(* CoDeSys 2.3 project: cy-wg-018-00.pro *)
(* Title: cy-wg-06 - ClevergyAS *)
(* Author: Andrea Ravasio *)
(* Libraries: Standard.lib 2.12.10 14:48:34, Util.lib 26.9.14 10:12:46, Visual.lib 2.12.10 14:48:34, WagoLibIdent.lib 25.2.13 11:12:16, WagoLibStatus.lib 2.12.10 14:48:32, SysLibFile.lib 2.12.10 14:48:34, SysLibRtc.lib 2.12.10 14:48:32, SysLibSockets.lib 10.2.11 09:20:54, SysLibEvent.lib 2.12.10 14:48:34, SysLibPlcCtrl.lib 2.12.10 14:48:32, SysLibCallback.lib 2.12.10 14:48:32, mod_com.lib 2.12.10 14:48:32, SerComm.lib 31.5.11 08:54:36, Serial_Interface_01.lib 22.4.13 12:50:14, Modb_l05.lib 22.4.13 12:50:12, Ethernet.lib 2.12.10 14:48:32, MBus_03.lib 22.7.15 16:25:47, WagoLibModbus_IP_01.lib 24.7.13 15:05:58, WagoLibMBX_01.lib 20.3.12 16:32:40, LON_01.lib 22.7.15 16:25:47 *)

(* PLC configuration (modules and I/O channels)
0750-9999/0545-0008 8 DO/DI Generic [Type_34_8_Channels] node 0, in %IB68 out %QB44 {INTTypePAAssignment = PLC; INTTypeModule = plugged}
  VPN_ST2 AT %IX34.0 [BOOLOnX_I] I 1: Digital Input
  LAMP_AL AT %QX22.0 [BOOLOnX_Q] I 2: Digital Input
  KEY_QE_ST AT %IX34.1 [BOOLOnX_I] I 3: Digital Input
  CIR01_EN AT %QX22.1 [BOOLOnX_Q] I 4: Digital Input
  CIR01_AL AT %IX34.2 [BOOLOnX_I] I 5: Digital Input
  CIR04_EN AT %QX22.2 [BOOLOnX_Q] I 6: Digital Input
  CIR01_ST AT %IX34.3 [BOOLOnX_I] I 7: Digital Input
  CAL01_EN AT %QX22.3 [BOOLOnX_Q] I 8: Digital Input
  CIR01_AUTO AT %IX34.4 [BOOLOnX_I] O 0: Digital Output
  CAL01_RST AT %QX22.4 [BOOLOnX_Q] O 1: Digital Output
  CIR04_AL AT %IX34.5 [BOOLOnX_I] O 2: Digital Output
  AT %QX22.5 [BOOLOnX_Q] O 3: Digital Output
  CIR04_ST AT %IX34.6 [BOOLOnX_I] O 4: Digital Output
  AT %QX22.6 [BOOLOnX_Q] O 5: Digital Output
  CIR04_AUTO AT %IX34.7 [BOOLOnX_I] O 6: Digital Output
  AT %QX22.7 [BOOLOnX_Q] O 7: Digital Output
0750-9999/0400-0008 8 DI Generic [Type_1_8_Channels] node 1, in %IB68 out %QB44 {INTTypePAAssignment = PLC; INTTypeModule = plugged}
  CIRD01_A_AUTO AT %IX34.8 [BOOLOnX_I] Ch_1 Digital input
  CIRD01_B_AL AT %IX34.9 [BOOLOnX_I] Ch_2 Digital input
  CIRD01_A_AL AT %IX34.10 [BOOLOnX_I] Ch_3 Digital input
  CTL01_ST AT %IX34.11 [BOOLOnX_I] Ch_4 Digital input
  CIR02_AL AT %IX34.12 [BOOLOnX_I] Ch_5 Digital input
  CIRD01_B_AUTO AT %IX34.13 [BOOLOnX_I] Ch_6 Digital input
  CAL01_AL AT %IX34.14 [BOOLOnX_I] Ch_7 Digital input
  CAL01_ST AT %IX34.15 [BOOLOnX_I] Ch_8 Digital input
0750-9999/0400-0008 8 DI Generic [Type_1_8_Channels] node 2, in %IB69 out %QB45 {INTTypePAAssignment = PLC; INTTypeModule = plugged}
  CIR02_AUTO AT %IX35.0 [BOOLOnX_I] I 1: Digital Input
  AT %IX35.1 [BOOLOnX_I] I 2: Digital Input
  AT %IX35.2 [BOOLOnX_I] I 3: Digital Input
  CIR03_AL AT %IX35.3 [BOOLOnX_I] I 4: Digital Input
  CIR03_AUTO AT %IX35.4 [BOOLOnX_I] I 5: Digital Input
  AT %IX35.5 [BOOLOnX_I] I 6: Digital Input
  AT %IX35.6 [BOOLOnX_I] I 7: Digital Input
  AT %IX35.7 [BOOLOnX_I] I 8: Digital Input
0750-0464#04 2/4 AI RTD / ADJ./ HA [Type_44_4_Channels] node 3, in %IB64 out %QB40 {INTTypePAAssignment = PLC; INTTypeModule = plugged}
  S01 AT %IW0 [INTOnW_I] Channel 1
  S02 AT %IW1 [INTOnW_I] Channel 2
  S03 AT %IW2 [INTOnW_I] Channel 3
  AT %IW3 [INTOnW_I] Channel 4
0750-0464#04 2/4 AI RTD / ADJ./ HA [Type_44_4_Channels] node 4, in %IB64 out %QB40 {INTTypePAAssignment = PLC; INTTypeModule = plugged}
  S05 AT %IW4 [INTOnW_I] Channel 1
  S07 AT %IW5 [INTOnW_I] Channel 2
  S06 AT %IW6 [INTOnW_I] Channel 3
  S08 AT %IW7 [INTOnW_I] Channel 4
0750-0464#04 2/4 AI RTD / ADJ./ HA [Type_44_4_Channels] node 5, in %IB72 out %QB40 {INTTypePAAssignment = PLC; INTTypeModule = plugged}
  S09 AT %IW8 [INTOnW_I] Channel 1
  S11 AT %IW9 [INTOnW_I] Channel 2
  S10 AT %IW10 [INTOnW_I] Channel 3
  S12 AT %IW11 [INTOnW_I] Channel 4
0753-0648 LON-FTT [Type_55_1_Channels] node 6, in %IB80 out %QB40 {INTTypePAAssignment = PLC; INTTypeModule = plugged; DataStream = 1F8B0800000000000400ED5D7B6FE2C8B2FFFF4AF73BF820DDD5AC14261808796C921503668296470E8FCC8E6646C88106BC636C8E1FC9E47CFA5BD56D1B1BB71F0498248CA5D52CB1DBD555DDD5BF7A74B97DF9E78F852A3C10C35474ED2A27BE2FE404A28DF589A2CDAE72B635CD8B95DC9FD7FFFB3F972D5D6B6A1631A6; DataStream = F29808F090665EFC3095ABDCDCB29617C7C78F8F8FEF1F4BEF7563765C2C14C4E3BFDBADFE784E16725ED14C4BD6C624E73D35497E2A27DC1AFACC90174D687C5EB828142E4EE1DF938B827851A85C14CAF02327FCAD4C3BF2825CE5DAB6A68C95A5A2D78949B4FFCA9A9E13FA449DD6F5B1BD209A255B205E4D5FE0EFAB5C; DataStream = 7532119E74DB10C6EC8A302706B0D721B6A16B0DC5583CCA06B9F3C6E49C76D4971FC8AD6CCDAF72B58BAF4313EE7E95B58941E4F7AAAC68CA57E8F9BBA52F73425B9FD82AE9D88B7B62C0D339183C41C0E16BCBC6F7EEFD3F646C99F4DAFA55E7225C1E90C552952DD29C0077CA542186770FEEE2C83427D78582C0FBEFF2; DataStream = D8B9EF7BA23FD697E41A6EB11FBE3B7F9127BC8EFFF35D6D6A13F2E35ABC3C663F3CBE8E6318F398C619B9EE376E079A3E214CB2D583F4A6F708B769B049D750668A26ABDCA6819BDE234DB3A58FBF93C9B565D8046470FFF43568C3D4C9966E3C796D56577CCDBA4BD41B59BD9ECAAA499B7957BC566D8213CDA61B8732F0; DataStream = B7D74A52096A5A4DB741DD60DD5C688A7A95C3CE73C2B16F4088F5A81BDFEF644391EF5562FA2765ED9EEF5692C63C4F6BE235C7D39EF3E2BAFAF854086F067528518F38BAD4B91B8CF4FB7F4606F98F4DCC286D5A6994F6A0F4DCA6E12601A5F137E56A532A8DDA40ABD26B5658BBC408EDA22DD3691823AA687DA24D06CA; DataStream = 824EADFFCF603BF947A09DEFCFF5763D3226CA03F135F55F5913FED6507443B19E56C27B57022DFBC47850C664F0049A571D7FD7F447954C666402DAE8BB1378A4AE18800C3090D74D6D69C3A4AE2E0459060B3755C63837D71D5D0326FC57024D6BBA365566B6416D08AC9225312C8598EB83DA34BDAED69465FD7AE0B10F; DataStream = 4F16E92BFF25D7A5CB63EFB76FD51F472FFB578B08A5384428ED1211C0B3B06C330520E87DA765221E782D5F3D1C143338480F075DDB7A5B785039183C388DC383D39DE1C1545109BA0869DC8306B4ED61D364F7C06BBA433CF0143D19105C9229F0E024C383C3750FC4E2E1E041390E0FCA3BC583F40E02AE7334FD695C84; DataStream = 55DB570F0A950C140ED849289E1E0C2A9C87D2506C8458D450D8292A2CF53490404DFFAD9E266858357DF580709A01C2E17A099B060DA13BAB8C6322CB97C7BCECF5F352DAF109EABC1891A1CE6F98A2A68BF24E312C5B5685A9AD8DD96A11EE5518D4F5CCF34669E498B59AE591D3E1FFEBCB2343F3B479E430ED1486C0D3; DataStream = 861D5A824D1248515A465B66A640786DBEA1275E96516623F4721965689D32A31CA29C01C36101C3CBFB881BE2C2E16496CFE23249673BCB2459A05AB87C17CB34B8808AD827295D063FE90C180E0B18DE9EC77038D9A4B3B3386438DB1532C8AA6C2CD2804295354C03090ECD0C0D0E0B0DDE9C9B503CCFD0609F6890DA47; DataStream = C800E12001E1EDB907878408711985B39D651430E627A9F28CEA539FB54D83080ED90C110E0B11DE9E8B7030782016E25C047A773788307F90C7A3853E49850A37B59A3882594E9F4FF091CFD0E1B0D0E1EDF90B62060F3F071E326CF8C5B1E1CD790E87040D27B1D070B2B35D08B8324AB5034171019BA5DF86706867B870; DataStream = 58B8F0F67C86430A295E2F3064A8F02BA3C29BF3163250D83728F4EDE53203865F1D183277214B313883B40287629681CCE0E18DC2C321A5195E353C64D8F08B63C39B8B290E091A5E634C51CC3290192EBC459FE190428AD70B0C192AFCCAA8F0E6BC850C14F60D0A5906320386CC5DC8520CDE20ADC0A1946520337878A3; DataStream = F070486986570D0F1936FCE2D8F0E6628A438286D7185394B20C64860B6FD16738A490E2F50243860ABF322ABC396F2103857D83429681CC80217317B2148337480E38D46F3E6509C80C1DDE283A6459863DFA0D080DD5B195790DBF3A2E64E144060B4158006FE15657B42CF9F84BE3C2DBF3173260D83330649B12192E64; DataStream = FEC2CBC1C2791C2A9CEF0C14CC47C51ACFD38042AD51476F41D27094521E00E910CF60E1B060217317325C08E0C2C70C17325CC8DC856C4FC21DA4A0CF90153E66E0F0069D866C4F628F390684866C43E2570785CC63C83021E42E641B12BF3C2EBC3D67210386FD0343E62FFCEAB870F0FE42E88EB9BA95C4F3E5714BD7DA; DataStream = B2F1BD7BFF0FB046AFAE5D33AF2FFFF5A556AF0EAA5F2EFFFCB1508507629840ED2A27BE2FE404A28D61C0B4D955CEB6A679B192FBF3FAB2265BB2AACFAE2F1B8A4A84A609FFB3884126F0484EA8C3CD3B8F44196960339CC2AB1CFE0B7FEBC642B6BC46156CD396FFD10DDF7339E156B6E657B9DAC557442D435E5032A6F0; DataStream = EEC759E5F7AF20C2271812F32B5234BFF607D54EBDDAABBF1F7CBE852729CC5DE522703027F4C814F8D5C624B615AA741FBF700BFC148FC5D271B1201605F1ECA258B8108BB9EB75B4A6AC70AF0A1F64D319813EACD4B1F5A5F22D27D0250CE2E7040A9E57B9D3524E4058BACAD18135C87F6C625A70EDC1620F238E8184D2; DataStream = A83FE80D6B0326290C0D8CA632664F52AC9BC2E323783C27A09621FB3961A829D0D96FAAF547537B90556522989601130BDD98BA6D8CC96F33EB0FBE503EF625CD5E082E79E46E64E1DCFD5016F6828A0220C37EE74557985EB41C5267D8E649E189DE57669AA3588E28AE2453DF10091A3C65E604E48EB0C5E00CE9098262; DataStream = 824C43CDA4BD804ECD602ECCA666911931685F4DB33FC6CF18D23F56729E9C944E5CF1684F3CE1869D7EF36347AA8F5ADDCEC79CD09D4E4D62514261811546043B23559FB8C580B84EAB7D4BE440BA60C102D06DEEC445C856E24F262537F2C8454BB950545531C958D726662A3961A6BF94566BC95B4075D00AB0F2A80982; DataStream = 3C99808E9B7C319ADDCE8AFD131EFB13D4728F0663F8C465D8C521AF9394EBBFB8E2B9E8F25C6524040B1F03E0B58CA7B8B51FCB34B263B9DC965C6E793DA4D5A5FE5C478A6994A954F2E140A914928F1A81189DEADF747B49023222214DF2E0E12C7FAF5882ED302F00E2310769BF2B2738C0CA86C85079163288952851D7; DataStream = 1D07EA463DC73E39A6C5BED78895D7F409895B53A9F4D3D4A29792C9E9670F5A2AFA94547C4B3AFA41B1BCC95913C8013F7D212B1A8FFD0FCD412341DF26CEC3D16C7B13C59A6E6C958453818A00FFF86CA223D0A95FA0E2A92B520794E1990269F4D16871A89E6934D2DA4488724888B22744D92F84CFAC02DE0A636C922C; DataStream = CA29DF92529B10230B1543D0A7023655483A23FA6C890686AC99320D79A8B36024CB75C65D283F46CEE3D1A2D106307A30599B82F906A0503C3909C2DD262070CE453A874CB464AC855F05B700EED36FFEA5C458F868E8F6726BC89E2DA3217B16E8616B004B42E1A04A3D0B7BEF755D25B2B60FD8AAAC5408FA7C26FF267D; DataStream = 340508B3A167CD7F79D3C1F8186AB6096DA70A5127CF14C5A624E244498AA4335392999200006F6D49668CCA762AC9372DCF3138CF73B91D80B7AD39EE098C5984AE7311276A70C40237E20592233D167D36C7FCE7C8E6E6B837958A9B175A02B10DA4DAC271287FF3AF503723590E64244D4BB6EC580F222E21E93EEDC4AF; DataStream = A7BBCF49B21E02294951E4E624FB919244A52457DCC7662459B3E8846465FF49888E87DCC85144DE2B7D6A921982913E1D39E4A253118E41DAB7807DA292B1452DBC1A1FA5A7C84E9A0EB11123B6B30C2C662663B27CCFCD46CA13C3E36C67597D07022212A96343595A3AD720A70A1C263E12BBE6BC6A18F2D317B1F20DD5; DataStream = BDC16668AA0B325E1608DB2A5D79BCB8D562D2477C78ED3DC513B0DAEB553F27C847A187117010A1E28AC7F800D6C48A309ECB063838C4489124A6ABA3060FA4B43D08A63E942B9E85845B1F12CE5CB22553BBA9F6560217B9B6D693F88B78F26D6DCD44A1234B7655FBB566733514CF375AB49F7FDBF224A53326964FCB67; DataStream = A54AF93429367386E1DFC36ADD370C5C64E4C4686BD2973D23FD646DE4413F1319074969CB20201637099D53AFD99D3A2289A0997A3BC4B77D73BE5BF861E8C34267A1598F401F2EF8780F3D177C58203D5226AE6C61ECA9084CFBF61BE3448ABFAD63EF49F8258435E9B2E93F29B8A9AC8D844AB49935DF3E0470E477C945; DataStream = 0F80D411C4F279E12C2FBAE915F799579729C58284DDA44A771FC7256F3A444AC5753037DD7FD82442DF026645DF169FB8AA41392BF94324223C80731CEFFB45847C180811CE6625BAD0CA8332B16555C0054BD7E90E72C68C5DA458884E1D857985070ABBC91944272613F81537E457DC0FBFC5B4FC1637E4B7B81F7E4B69; DataStream = F92D6DC86F693FFC96D3F25BDE90DFF27EF83D49CBEFC986FC9EEC87DF4A5A7E2B1BF25BD90FBFA769F93DDD90DFD31DF29B8EC3B3E4643DD7B58167CF5E187CCF9FCFFAF90BE3B01863E8927817F764F45283B21863F51299DF93054C8DD0628C094C647E4FE630355C8B31F63091F93DD9C6D4D82DC618C744E6F7642853; DataStream = 03B918632913994F6D357756F5E746045E16060BE2718363C1DDCB4C880770D375E43CCCB8F736809E886C1C090B5DB3E647C2447E3A12E6BA8D5714CDB6C891C00A8253664DD367CE4A05ACF2E76C0E7D26323FE2F1E7D0C2623ED1C7E2D28145BFC49BA403378A5F5D31DA38A09BC4AFDCA07CC1A844EB1E6DB027614AAB; DataStream = 4499CC2D868E12851B894FE4D88A07B8BD27318A5E507D038ABD891C659E1C734A245A10BCBF27494ECE3DEDA28B73EB1AD985432646BF688BBDCBD36720B3813CDCC22107ABE27258BED71BB6C9DFF8F2E4E26AC7FECCDBFAA982B08BE76FD9E3582D3CE0DA4BC6BCA53BF51F1B24CCDD6762F2E5618154EFA197CD914709; DataStream = BCE51A72C5DB2C418E026F9D1F7FE63E157BF53062DB6393B723744A886D7F446E58B146A9F7EE693D0955FF116E8505CA494AC580C7500A2E362B62FB8DD594C4D6ADADFA8BDB4495BD6EA22B4C4ED38AB8740A95462A79206A9AAA19AFB4893E912C29B78C2DD86D9CB4CB4077D1129FFDA497FC10283A779BD4D37037B4; DataStream = A81E8E2C7D84381BA7B7CAAA53612CDB2682AD03CB89F2329C2D539CBDC3147B04C89679207BC7F6CE127724F9DB38CECEDBDA0EB807B5E59F02B55C9937D8CAE1022D958C96C9C484623F17565910131FB744692717513951CC1B085D442EA8BECDD845E4C2E61B0C5EF8C5436F347AE19700BDE1F0A5C8DF83DF287ED935; DataStream = 9A9D9FFB66C87B157C938A266EE0BFF0D3DAD9DBE77E13CBFC3F55598087BD81A1F53D96C2DCF2CBB598E7E8D07859A31B330A1BE8658C7F4C496F6780B708B983E5BC8EF379EE995F5A6BB9D44D252A3E4D53240FCF87A2D4259E7E468C23B79E67FFC5913D224F8E3F81EF8D02D1CE134B2539AF183D8E96564246D4D354; DataStream = 5A5D8D53B77A4F71FFC75C7842A6A8D50AE20C372F07024756697920B37AAF6A5513BA739DF41C2927D07EFE5132103B8F7CA7B1048E9368D68F3CCAAF2861F013B3040E61DE5938C53237844E9E906008CD35D2C16EE342683DD05D74088D91EA968AE8DB3C2AAE768FCE4B6B923F3B21899A187C85A8E25744E7C59BA92A; DataStream = CFD29BB983D1C6C4620D27679B6FD6E910256F4472154F6154F8BCEF602B554C2784ABCE3B9064B5867E7E29475D3191C8641B39260E8D1729E7E8DA565E9FE6A957666E23856E5BF8821923F422C51DDD25D1F263C518DBCA567AA5039D9143E7450A3D9C3931D9C9893B981487D28B147EB4C9782E6B0A749C9FCAB6BAD5; DataStream = CC2C3C5A234AEB458A411A844CEEE5F1771047516D63ABF9993AB4460EAD9F54F6D77D2046DE90B5595AE6B921B90E544694CA8B589221D8D51D486123997D8A916041247C77D5D8787D7065211EAD7DAE8F048B32A4DF0CCA5B7A7E416433FD0289981D24863B2D0EB117B12C357DB1B035E7A80373C385CF956B0C14F7B0; DataStream = E8D3DB9806F44D266063D469DE4AEF887185413946486964EDCD0F4B2A2F74E5C82B5A7E891CE2E1435BC8E4893352B4914BF045EC0D3B89380FA67C1B79544A65C43FBC731F36A62D6B3660DA58D72C435753B2CECDC92C28A59143E985A29625F8646CEB7E0B494095DC9A9C9F6F68980C68B40D659216BCA2C470C9BC88; DataStream = 85E991A56E58F9856C7EDF460C839219219917B12A2E478A36CBE3D7B1B69165B9A245BFB4F52236C52F10DA845D0984B45EC4AAD0CD90BCA65BCAF4293FD92CD4E74AC5B64018C1D17EE3FE04ABD22326FF7DDF540B07EE011E2F962A89DF397DC6117D6782DFB478A590D8A7F14026295EDBE06EB1F99EDFC7E95B5B24FA; DataStream = 57EF60D30F683E23AD6A3A0FAEE51F69A90BCBAA92BDEC1AAECA5622AB8DD67708A34B8D9C4971DF91F8C032EE6B13F47FF448245B55DDF2B544BDEA6F73A670F0B0A9B8B346D6EB3FA28E9F4A386CC41394B6A5E7DB6D79BE8A931E77B7084E5216BE144F2B81F3688AA725D1DB5AC42FB6E0DE038D5D367EC7C2F72997E0; DataStream = 60B8D35E8C7BED6242C01327A65023AAA9D869B618E92E0FFD04A5E51B88B3802273E7FCE6AE5A1316110708449D3116FCE065DC147BE463B674CA91B36F5E5FFADA07FF12565F4E18C833E7AC9FD506D7F525ABAC0B24E405670987256AF4469D612B27F4E447DA860DD171904A1FA96B9622AB823C1E63EC6510DCBBE692; DataStream = EBDE4A9DD1A03BEA4B9D7A0A4A8FB8BF9B40AA27D5A4E69DE4E732CC644DD54D22C81A80BBFC409CA3C7B8646BAD6E5F1A359AAD00C5620CC509415B984CB32EB5A44198742944BA478FEC043627F49334BAF1E47E4F804BBDDE842118747B9F61DD75FF1ADEFA8997C3C481657DB1E1548D7A553FD59304AA1B4CDB1A6576; DataStream = C0DEB14FA3B9EA5DF1ABB7776EE0A6DADD4FA1DDB42CC4C2E34DA7C4104C9B0A08662882E0DF0D0944FC2B44A6EECDA4AAEBDFF1C8DF244A6C2E29AD38C5960C4337043C85734934F45A22D5B0CF86BE516DB6E235DB233959633A9E53A9D78B57EBE0502A9AB0CAAD448FE5B053977A9FB08E2A4EA93D96519F61148E5103; DataStream = 1346A3D95D6739ACD64196F125C88940F3285C8A83665BEA0E07EB642B21B29F14582D8F8249F16E4C0482EC4710FDD4ECD4BB9FD6699E8668AE1DCAEA2518B944ABC3C1CD3AC9B33049B69A99A1D22DD0D92586CD848F1840B55693FA7D98B2EADD9A929D2700C63D79D20149A52EF7540420DD97A4BF46CDCE5DB585DBF6; DataStream = BE055108CF99D3FA53B5C9F53A83F77DA4C474D873EA604FE01D93200BC3E5047D386F7EE7A095843BC1D5D6E846AA828A076128BC78D6494E75DD8A24D9E87607EB24C3EBBC4EEEED193D5E103FE88512BEC3599635F69AC2EF11C4EBD287E1C720ED302C357D546DC67A2AE2CD4EA31BA41D9EE0FE93093EE4E68CF73FF7; DataStream = 07523BDC45787D0EE6CED9D282620A4EAD410451D0C8A1C4D3CC7C184D02646570F135305D9A7388523A196ADD0E7E2D2DA0B8F9301E624F1342B790A12B7D3A55158D8B0540B2DB68B49A9D804B920FEB1F2B0EC5E25A854DAA865FFA83915FC84FB07C8509B4B4742A956FC3C4852101D0792E1B934719F74ED8B5281187; DataStream = 9DBF3ADD4F9D003F61E575ADBBEF9D2A6718E5354E29722DC9183F613989EA34D911E8E8C23AE525661634AE3540925D9CAD7A73408F855D5FCE9AC7D28664ABADB69F6E9C6F30D02D593D766B096821E803FAD6B43F517887691C5D83AE688519187B53701BC37CE1197416D164409BA8511B7407A3FE5D8DF224C63B15B1; DataStream = BC7037C8D7E817E39D8B58FADC6D9135FAA5780FC3298E06ABED1448B34953896C08DC901FC8B7C06EB7DA0370FF7BC1E10943431CF9A8D1F1932FC63B1C8CFC5C99CD3760FFA6F9F186CF3FC7FB88EB204A804007C5045F843B4049231F52CCB023C2279C34E6218DE4D8A98831491CEE10D31CFB1A413B71A4C37C87976A; DataStream = 0390601D94A21C8D660F490608F21C7F2008A8964F4FF4B627850887172512CE1B04BF353C01375DB7EFC15D7F47EB1F7E4FD5CDA0F72180FB222F04F0F5011E30228CA9D3EF77B880FD8EBC9FBD3F02236328DA77150205447033C6C461D7FDE1ED5DA0EBF0AA0D8A873BDCD4154F3F8A03A93F080D6378F146F4B3D98CD1; DataStream = BE78D3165ECB81FE162C152710ED4131740DDF3701DC46D34434933911EC056208EDC6737EECE1B02075EE6ADDF6EDA85DFD3BC04178D1073890EF35742455B01A4BDB4A256CBBDB690EBA3D6A8803768F138E0485F56C2A4C2331A28C3CEDA3DAECE0EC49BD80B757E4E428F08BBE82BC5CAAAEDB15195022EDEA00FE85E0; DataStream = AF1B8CD7C3AC7721A23418ADC45109D30BF3C9E8810F48131549143F557B9D66271069948AE942B43327440BBD23BF6186E8364DFEB3A53F62110D5B29CBB577ECB9345BD29DD41A85C7DBBBC53511FEBB715E9FD78E6B0CFC77E3FCB51B302DCF12AB14EFA7B5942911FAF29400316A17A8253385771FAA353C1CD83BA4A0; DataStream = C805CFDB354F246C136ED977B49F5275528AEAA418EFAE51A27D9F3160F63844BF1C45BF14EFAF51FA0366D08E1BB436F05D5D3197AAFCF47BB89793A85ECAF14E1BEDE516E089727F24D06D891A66CEC680271284044B84E328E12A51DD56E25D39DA4DD48C9C45113D8B77E3A278EF0D3A474C07E057DC208A8548852B24; DataStream = 387AB46F4A5E6558E02E175E3791A32656383E5F22D4213B14EB422F336D8875BD7FA7C03A89D6643A2F4ED1CD0F832CF407B8E21505F129777BED6A8B9315377DF4229EAD37FBD50F2DA91E8F7AAC30C8E5CC7DD3884B70785BAF0E7067BD3A18F6E351F096189864F2C8BAA5861194FB52AB411DA1780C74727972E088A7; DataStream = 3856ABAD6AAF1D0F7B8EFCCE7B547854102B6EE292ED49B7DDDE003C8CFE5FF138D7754BC66267A87B07D6BF5997E2312DA03B1194A40E4E753C6AF51C8D635392A078BDF61D97BD302AD568A89A467F6A2DA9DAE3A84F189402349DF2BF1892A169E6608D338A4C77683591E29E8EC5A54C69C2FA1B341B9F9DE1AD737086; DataStream = B72A9FD70777B9723699024832A5F926ACF514BC5A4F6E57ED6A678869D0412F18B7851759B803842A5A5911D7414F6A7761C5853AE0EC39B10E7CD56A58A142D37A4C8CA932B31DB05E32A7847E8791DBED6DAFFBB1570D4E7E7839327DA2355879B7068BD6A409EF8285595C1BE3E9594FEA4BC1AD0FCE6AFD41C6365067; DataStream = 9D79DB0E2061EC020E930E2F60260540A02CA8FA2C96D35637E0FF7362C9962E43CC3AF7E66195EAC51DC67EED768037D837C722BA6A75AB75EE047076AD6C8D7636B60D03BC0B157746E509F4E5F4FE5E684E03DC3CCAA630975516FBA17EAB4F47D04031854745C598D6048B2E18B6C6F66E0D7DC11EC7D7F63175BF7AFE; DataStream = 7DD4880F3B3CE63991E80DD049E07EE071B674AAE682634B4B93D0ECCBF89D77A615E063C1A860DA1F6FF8C5F23F4A457B84F88F08609B92C5BAA9B6065CB978A61FF832E2455B0DED3D992974B4230714EC77B5C7EF3C8C63434D753530AAEF28DBDE8952BC2207CDD8723469471AF961E1D2A1AEAEBE743DC277B8C9E314; DataStream = FDA1EF7B042BC0A4E58770F7883D20DCE3DB004702B1C6EF7FC7D59CA40FEB93BFB0C1BFBD27C26FFFB175EB0F65A212F60B770CD82F36AFCE55DC121A8FC9D2624AEF68C991A0632AE051319936A0CE004D65A6E906A844A05B8358B6A199488943DFD1C8A985890A3A46F48BA4D3407751DEDA40BAE50E7F39A5EB5D765C; DataStream = 6FA7C28CEF703F4439DC1835A470B96BCC5C615A51B62D9D124018C1CFB06933827BE7D623215A20FF83F93BAEA9A19D5687836E181D884C2B26744DE5161AD1276FA4EA20DE0FAFAEB8C83B503C067658CAE7116BAAF97524947CBBD7F938FAD46B076B9838B557BAAE26F25AEB765BF17E3897574D99CD2182B38D59CCAC; DataStream = 353FDE00400C7B1FA578AF9CDB03E655C73ADF03A1E4318BBACE3DC7195829066E713A6E0D1B17DB5ADA56B402741B8D045FDD8B9FEF0912C498879F7AA5F4D6439EB0CD9760F1CCC08378C25A088B9594BCA33F97F662C975572865A92DF53E86D48EB33DA478A3C0928A0440662A83B506F0C0A21DAEEF4ABB68543BA36E; DataStream = A7F539C1957754EE51B1E6343B8D297E9D75EA98EFE81E7A52784239BE7D734CF20BF93B76C32A4823E8356B52820BEFD4B7D2C14E24D7AEFE1D5ED81C8F1DC6565F80FE22521CE378C493956ADD4EB7FD39C14DAF93B9BD50265E88114FB32EDD0CDB6B1540E1555703E0BD375290AB555BCD0F3D88B013FCEE95F68E93C5; DataStream = A61A1B9A6DCE1AF388C2DA024397822A58AC6AD2668E37A58C8598390FF1C84FD58D6EEE6AD4478EB60A5E8358E7994167379E96773FE4CA06EDF171B004FA182BF5AE2F69BD5ED384FF8143E0D45ED721D0B82386090D515BDE03356CC68ABA1B4B880A1AB48EC86B73824DDAF23FBAE17B0C1896AD39E8D6C55787734AC5; DataStream = 14DEFD38ABFCFEB5A56B9F74E3BBF99516687FC51A9D7AB5577FDFB8756AD09AC04CA120F0FE0359C914D885F82AB6157EC0A18F9F60C0E5792C968E8B05B128886717C5C205AC5790DED6A8AF27ABD023FDDC33E79AE7BDB8B5EEF89D3CA1EB05758A365696B21A716A411F04C24FDE39ED4305F830F86DF0B864AC1A65EF; DataStream = 15103C308B7DD4DAD7E9FA414AE19EB407A5E7DEC541F51D8E15AEFB4FE876FD40ADE8F48EF6A0BB1F17F7775AE2761AECC47B99872A61BC64D804A40B74729AA6934AA0935839B005CA12ECA49CA293D34027AB33F12245B9D5D7C6CB59B121E5E35D5BADDEE31A6E64EAB3EB6FDFE08F16BE0B01CB782A8FC9F5FF035C4A; DataStream = 7264312E0100; DataStream = .; DataStream = .; DataStream = .; DataStream = .; DataStream = .; DataStream = .; DataStream = .; DataStream = .; DataStream = .; DataStream = .; DataStream = .; DataStream = .; DataStream = .; DataStream = .; DataStream = .; DataStream = .; DataStream = .; DataStream = .; DataStream = .; DataStream = .; DataStream = .; DataStream = .; DataStream = .; DataStream = .; DataStream = .; DataStream = .; DataStream = .; DataStream = .; DataStream = .; DataStream = .; DataStream = .; DataStream = .; DataStream = .; DataStream = .; DataStream = .; DataStream = .; DataStream = .; DataStream = .; DataStream = .; DataStream = .; DataStream = .; DataStream = .; DataStream = .; DataStream = .; DataStream = .; DataStream = .; DataStream = .; DataStream = .; DataStream = .; DataStream = .; DataStream = .; DataStream = .; DataStream = .; DataStream = .; DataStream = .; DataStream = .; DataStream = .; DataStream = .; DataStream = .; DataStream = .; DataStream = .; DataStream = .; DataStream = .; DataStream = .; DataStream = .; DataStream = .; DataStream = .; DataStream = .; DataStream = .; DataStream = .; DataStream = .; DataStream = .; DataStream = .; DataStream = .; DataStream = .; DataStream = .; DataStream = .; DataStream = .; DataStream = .; DataStream = .; DataStream = .; DataStream = .; DataStream = .; DataStream = .; DataStream = .; DataStream = .; DataStream = .; DataStream = .; DataStream = .; DataStream = .; DataStream = .; DataStream = .; DataStream = .; DataStream = .; DataStream = .; DataStream = .; DataStream = .; DataStream = .; DataStream = .; DataStream = .; DataStream = .; DataStream = .; DataStream = .; DataStream = .; DataStream = .; DataStream = .; DataStream = .; DataStream = .; DataStream = .; DataStream = .; DataStream = .; DataStream = .; DataStream = .; DataStream = .; DataStream = .; DataStream = .; DataStream = .; DataStream = .; DataStream = .; DataStream = .; DataStream = .; DataStream = .; DataStream = .; DataStream = .; DataStream = .; DataStream = .; DataStream = .; DataStream = .; DataStream = .; DataStream = .; DataStream = .; DataStream = .; DataStream = .; DataStream = .; DataStream = .; DataStream = .; DataStream = .; DataStream = .}
  AT %IB24 [BYTEOnB_I] First Byte of 24
  AT %QB0 [BYTEOnB_Q] First Byte of 24
0750-0478 2 AI 0-10V 16 Bit S.E. [Type_8_2_Channels] node 7, in %IB88 out %QB40 {INTTypePAAssignment = PLC; INTTypeModule = plugged}
  VRD02_ST AT %IW24 [WORDOnW_I] I 1: Analog Input
  AT %IW25 [WORDOnW_I] I 2: Analog Input
0750-0478 2 AI 0-10V 16 Bit S.E. [Type_8_2_Channels] node 8, in %IB112 out %QB64 {INTTypePAAssignment = PLC; INTTypeModule = plugged}
  VRD03_ST AT %IW26 [WORDOnW_I] I 1: Analog Input
  VRD01_ST AT %IW27 [WORDOnW_I] I 2: Analog Input
0750-0556 2 AO ±10V [Type_14_2_Channels] node 9, in %IB116 out %QB64 {INTTypePAAssignment = PLC; INTTypeModule = plugged}
  VRD02_CTRL AT %QW12 [WORDOnW_Q] O 1: Analog Output
  AT %QW13 [WORDOnW_Q] O 2: Analog Output
0750-0556 2 AO ±10V [Type_14_2_Channels] node 10, in %IB120 out %QB64 {INTTypePAAssignment = PLC; INTTypeModule = plugged}
  VRD03_CTRL AT %QW14 [WORDOnW_Q] O 1: Analog Output
  VRD01_CTRL AT %QW15 [WORDOnW_Q] O 2: Analog Output
0750-0650/0003-0000#03 RS 232 C Interface (Adjustable), 3 Byte [Type_21_1_Channels] node 11, in %IB120 out %QB68 {INTTypePAAssignment = PLC; INTTypeModule = plugged}
  AT %IX28.0 [BOOLOnX_I] Transmission acknowledgement
  AT %IX28.1 [BOOLOnX_I] Reception request
  AT %IX28.2 [BOOLOnX_I] Initialization acknowledgement
  AT %IX28.3 [BOOLOnX_I] Input buffer is full
  AT %IX28.4 [BOOLOnX_I] Number of received characters Bit 0
  AT %IX28.5 [BOOLOnX_I] Number of received characters Bit 1
  AT %IX28.6 [BOOLOnX_I] Number of received characters Bit 2
  AT %IB57 [BYTEOnB_I] Input data Byte 0
  AT %IB58 [BYTEOnB_I] Input data Byte 1
  AT %IB59 [BYTEOnB_I] Input data Byte 2
  AT %QX16.0 [BOOLOnX_Q] Transmission request
  AT %QX16.1 [BOOLOnX_Q] Reception acknowledgement
  AT %QX16.2 [BOOLOnX_Q] Initialization request
  AT %QX16.4 [BOOLOnX_Q] Number of characters Bit 0
  AT %QX16.5 [BOOLOnX_Q] Number of characters Bit 1
  AT %QX16.6 [BOOLOnX_Q] Number of characters Bit 2
  AT %QB33 [BYTEOnB_Q] Output data Byte 0
  AT %QB34 [BYTEOnB_Q] Output data Byte 1
  AT %QB35 [BYTEOnB_Q] Output data Byte 2
0750-0653/0003-0000#03 RS485 Interface (Adjustable), 3 Bytes [Type_21_1_Channels] node 12, in %IB120 out %QB72 {INTTypePAAssignment = PLC; INTTypeModule = plugged}
  AT %IX30.0 [BOOLOnX_I] Transmission acknowledgement
  AT %IX30.1 [BOOLOnX_I] Reception request
  AT %IX30.2 [BOOLOnX_I] Initialization acknowledgement
  AT %IX30.3 [BOOLOnX_I] Input buffer is full
  AT %IX30.4 [BOOLOnX_I] Number of received characters Bit 0
  AT %IX30.5 [BOOLOnX_I] Number of received characters Bit 1
  AT %IX30.6 [BOOLOnX_I] Number of received characters Bit 2
  AT %IB61 [BYTEOnB_I] Input data Byte 0
  AT %IB62 [BYTEOnB_I] Input data Byte 1
  AT %IB63 [BYTEOnB_I] Input data Byte 2
  AT %QX18.0 [BOOLOnX_Q] Transmission request
  AT %QX18.1 [BOOLOnX_Q] Reception acknowledgement
  AT %QX18.2 [BOOLOnX_Q] Initialization request
  AT %QX18.4 [BOOLOnX_Q] Number of characters Bit 0
  AT %QX18.5 [BOOLOnX_Q] Number of characters Bit 1
  AT %QX18.6 [BOOLOnX_Q] Number of characters Bit 2
  AT %QB37 [BYTEOnB_Q] Output data Byte 0
  AT %QB38 [BYTEOnB_Q] Output data Byte 1
  AT %QB39 [BYTEOnB_Q] Output data Byte 2
0750-0653/0003-0000#03 RS485 Interface (Adjustable), 3 Bytes [Type_21_1_Channels] node 13, in %IB124 out %QB76 {INTTypePAAssignment = PLC; INTTypeModule = plugged}
  AT %IX32.0 [BOOLOnX_I] Transmission acknowledgement
  AT %IX32.1 [BOOLOnX_I] Reception request
  AT %IX32.2 [BOOLOnX_I] Initialization acknowledgement
  AT %IX32.3 [BOOLOnX_I] Input buffer is full
  AT %IX32.4 [BOOLOnX_I] Number of received characters Bit 0
  AT %IX32.5 [BOOLOnX_I] Number of received characters Bit 1
  AT %IX32.6 [BOOLOnX_I] Number of received characters Bit 2
  AT %IB65 [BYTEOnB_I] Input data Byte 0
  AT %IB66 [BYTEOnB_I] Input data Byte 1
  AT %IB67 [BYTEOnB_I] Input data Byte 2
  AT %QX20.0 [BOOLOnX_Q] Transmission request
  AT %QX20.1 [BOOLOnX_Q] Reception acknowledgement
  AT %QX20.2 [BOOLOnX_Q] Initialization request
  AT %QX20.4 [BOOLOnX_Q] Number of characters Bit 0
  AT %QX20.5 [BOOLOnX_Q] Number of characters Bit 1
  AT %QX20.6 [BOOLOnX_Q] Number of characters Bit 2
  AT %QB41 [BYTEOnB_Q] Output data Byte 0
  AT %QB42 [BYTEOnB_Q] Output data Byte 1
  AT %QB43 [BYTEOnB_Q] Output data Byte 2
Fieldbus variables [FB_VARS] node 1, in %IB0 out %QB0
Flag variables [FLAG_VARS] node 2, in %IB0 out %QB0
Modbus-Master [MB_MASTER] node 3, in %IB0 out %QB0
*)

(* Global variable list: Global_Constants *)
VAR_GLOBAL CONSTANT

	Plant_NAME			: STRING :='cySN:18 cyVER:1 - ';
	Plant_SN			: DWORD  :=18;	(* S/N Impianto di telecontrollo *)
	Plant_SW_VER		: WORD   :=1;		(* Versione SW installata *)


	(* Colour defines *)
	COLOR_RED			: DWORD	:= 16#2020F0;
	COLOR_YELLOW		: DWORD	:= 16#20F0F0;
	COLOR_GREEN			: DWORD	:= 16#20F020;
	COLOR_LIGHT_GREEN	: DWORD := 16#006000;

	(* Parameters *)
	Plant_DefaultTAmb	: INT	:=100;		(* [.1°C] Temperatura ambiente di default in caso di rottura sonda *)
	Plant_MaxRunTAmb	: INT   :=250; 		(* [.1°C] Temperatura ambiente massima funzionamento impianto *)
	Plant_AntiFreezeTAmb: INT   :=-40;		(* [.1°C] Antifreeze temperature, start circulators *)
	Plant_VRD_TAlarm	: INT   :=450; 		(* [.1°C] Temperatura di allarme VRD, blocco *)
	Plant_VRD_TMax		: INT   :=430; 		(* [.1°C] Setpoint massimo per uscita VRD *)
	Plant_VRD_TDefault	: INT	:=300;		(* [.1°C] Temperatura di default in caso di errore climatica *)
	Plant_CirOffDelay	: TIME	:=T#15m;	(* (Def.T#15m) Ritardo spegnimento pompe per ricircolo caldaia *)
	Plant_MaxWaterLoss	: WORD  :=2;		(* [lt/h] Massima perdita del circuito *)

	(* Filesystem *)
	FilesPath  			: STRING :='S:\';

	(* TCP Logger *)
	Logger_SERVER		: STRING:='';
	Logger_IP			: STRING:='192.168.100.3';
	Logger_PORT			: WORD  :=80;
	Logger_GETSTART		: STRING:='GET /cygmsrv/hsgm.ashx?';
	Logger_GETEND		: STRING:='$R$N$R$N';
	Logger_CHECK		: STRING:='True';
	Logger_CRLF			: STRING:='$R$N';
	Logger_DataFile		: STRING:='S:\LOG.DAT';
	Logger_DataFileOld	: STRING:='S:\LOG.BCK';
	Logger_IndexFile	: STRING:='S:\LOG.IDX';
	Logger_ConnRetries	: BYTE:=5;
	Logger_RecoverMsgs	: BYTE:=25;

	(* TCP Remote *)
	Remote_PORT			: WORD  :=10;
	Remote_WELCOME		: STRING:='Connected$R$N';
	Remote_OK			: STRING:='OK$R$N';
	Remote_ERROR		: STRING:='ERROR$R$N';

	(* TCP Sockets *)
	MAX_SEND_TCP_SERVER					 : DWORD:=3000;(*60000*)
	MAX_RECEIVE_TCP_SERVER				 : DWORD:=3000;
	MAX_RECEIVE_TCP_SERVER_SOCKET	 	 : DWORD:=1500;
	MAX_SEND_TCP_CLIENT					 : DWORD:=3000;(*15000*)
	MAX_RECEIVE_TCP_CLIENT				 : DWORD:=1500;
	MAX_RECEIVE_TCP_CLIENT_SOCKET		 : DWORD:=1500;
	MAX_RECEIVE_UDP_SERVER				 : INT  :=1472;
	MAX_RECEIVE_UDP_CLIENT				 : INT  :=1472;
	CONNECT_WATCHDOG_TIME				 : TIME :=t#10s;

END_VAR

(* Global variable list: Global_Retain *)
VAR_GLOBAL RETAIN PERSISTENT
	Mode_Manual : BOOL := FALSE;

	GRU01_Clima	: typ_Clima;

	VRD01_Clima : typ_Clima;
	VRD02_Clima : typ_Clima;
	VRD03_Clima : typ_Clima;
	VRD04_Clima : typ_Clima;

	Ctl01_Counter	:	DWORD;

END_VAR

(* Global variable list: Global_Variables *)
VAR_GLOBAL

	SYS    : typ_SYS;
	Logger : typ_Logger;

	Lamp	:	PLANT_STATUS;
	T_AMB	:	INT;		(* Environment temperature *)

	(**** PLANT OBJECTS ****)
	(*...*)
	GRU01	:	obj_CAL_VT300GW2 := (ID:=1);

	(* Water counter (NB il peso è moltiplicato per 10) *)
	CTL01	:	obj_CTL	:= (ID:=1, Peso:=10);

	(* Heat counter *)
	CTB01	:	obj_MBUS_CTB_SHARKY775 := (ID:=1, Address:=1);
	CTB02	:	obj_MBUS_CTB_SHARKY775 := (ID:=2, Address:=2);

	(* Cronothermostat *)
	THER01	:	obj_CRONTER := (ID:=1, Local_MaxRunTAmb:=250);
	THER02	:	obj_CRONTER := (ID:=2, Local_MaxRunTAmb:=250);
	THER03	:	obj_CRONTER := (ID:=3, Local_MaxRunTAmb:=250);
	THER04	:	obj_CRONTER := (ID:=4, Local_MaxRunTAmb:=600);	(* There is no an environment probe	*)

	(* Hot domestic water *)
	ACS01	:	obj_ACS := (ID:=1);

	CronEd	: 	obj_CRON_EDITOR;

	(* Boiler *)
	CAL04	:	obj_CAL := (ID:=1);

	(* Pump *)
	CIR01	:	obj_CIR	:= (ID:=1);
	CIR04	:	obj_CIR	:= (ID:=4);

	(* Modbus double pumps *)
	CIRD01	:	obj_MODBUS_CIR_DOPPIO := (ID:=1, Address1:=1, Address2:=2);

	(* ModBus Pumps *)
	CIR02	:	obj_MODBUS_CIR := (ID:=2, Address:=3);
	CIR03	:	obj_MODBUS_CIR := (ID:=3, Address:=4);

	(* Valves *)
	VRD01	:	obj_VRD 	:= (ID:=1, ReducedRange := FALSE);
	VRD02	:	obj_VRD 	:= (ID:=2, ReducedRange := FALSE);
	VRD03	:	obj_VRD 	:= (ID:=3, ReducedRange := FALSE);

	(* Temperature probes *)
	TPV01	:	obj_TPV := (ID:=1);
	TPV02	:	obj_TPV := (ID:=2, IN_WMIN:=50 , IN_WMAX:=800);
	TPV03	:	obj_TPV := (ID:=3, IN_WMIN:=50 , IN_WMAX:=800);
	TPV04	:	obj_TPV := (ID:=4);
	TPV05	:	obj_TPV := (ID:=5);
	TPV06	:	obj_TPV := (ID:=6);
	TPV07	:	obj_TPV := (ID:=7);
	TPV08	:	obj_TPV := (ID:=8);
	TPV09	:	obj_TPV := (ID:=9);
	TPV10	:	obj_TPV := (ID:=10);
	TPV11	:	obj_TPV := (ID:=11);
	TPV12	:	obj_TPV := (ID:=12);

	(** Communication **)
	(* ModBus *)
	MODB01	:	obj_MODBUS		:= (ID:=1, COM:=3, BAUDRATE:=BAUD_9600, RS485:=TRUE);

	(* M-Bus *)
	MBUS01	:	obj_MBUS		:= (ID:=1, COM:=2, BAUDRATE:=BAUD_2400);

	(**** SIMULATION ONLY ****)
	(*...*)
END_VAR

(* Global variable list: LON/Module_1/InterfaceBlock_Module_1 *)
VAR_GLOBAL CONSTANT
(******************************************)
(* Automatic generated code, do not edit! *)
(******************************************)
	abSignature_Module_1 : ARRAY[0..15] OF BYTE := 16#7A,16#26,16#60,16#DB,16#56,16#3B,16#16,16#40,16#89,16#16,16#11,16#E4,16#B0,16#D6,16#83,16#3B;
	wConfigSize_Module_1 : WORD := 504;
	abInterface_Module_1 : ARRAY[0..125] OF DWORD :=
		16#1028C19F, 16#2137A508, 16#6041B800, 16#06246830, 16#428B2E71, 16#64B95263, 16#FE000902, 16#2A050140, 
		16#201E4092, 16#8BD6B010, 16#8102570F, 16#1890E46A, 16#5C1D0704, 16#D47157C7, 16#1D2B759C, 16#539D1D5A, 
		16#8D25581D, 16#286C1D4F, 16#65AAA48D, 16#A999312F, 16#3871E72B, 16#2E679A2C, 16#1526509A, 16#A942353A, 
		16#2CD9B76E, 16#AA15FBB4, 16#4EBA63CB, 16#244B36E8, 16#BA6FF382, 16#3B16A4DC, 16#65DBB67D, 16#16245DB7, 
		16#CBCA2D8B, 16#AE5B9800, 16#96959AD6, 16#DCB275E3, 16#980083EE, 16#D22A265F, 16#96EED4B7, 16#E6D6A51B, 
		16#B49229B9, 16#659BD6E8, 16#922C6495, 16#A68DAF9A, 16#146D324C, 16#0BF59CD9, 16#F0E6207B, 16#A95A0509, 
		16#0C30595F, 16#2A0F6A98, 16#1548A5A5, 16#2835283B, 16#CA0DCB36, 16#138125DA, 16#9097AD54, 16#7A002B99, 
		16#0E1D8A54, 16#A3A65F63, 16#E7C47284, 16#CB52452D, 16#EC15B86D, 16#A99847E4, 16#04176EDD, 16#5C8A4C1D, 
		16#1C5445A1, 16#988C80B5, 16#45CDF448, 16#437D14CF, 16#1908420B, 16#29D10D87, 16#8F957715, 16#BA63838A, 
		16#358C6C0D, 16#DCA67D0B, 16#50958048, 16#0943D4E8, 16#1BD66D51, 16#870EB015, 16#3DA1A3F2, 16#51472006, 
		16#6AD45591, 16#AD028665, 16#09DCFECE, 16#00010604, 16#EE3FC081, 16#1B047261, 16#4C28E600, 16#38E51802, 
		16#ED3602AC, 16#1EAC8339, 16#837136A7, 16#3520E7F4, 16#E020C09F, 16#2340A3D3, 16#88B153A1, 16#08783AC0, 
		16#784A0804, 16#5A040428, 16#0DD83178, 16#0133084F, 16#6B86E1E9, 16#28AE2588, 16#1AB2B876, 16#8E6B0BE3, 
		16#E640AE29, 16#E41A23B9, 16#41946BCD, 16#B9F658AE, 16#91E6DA84, 16#AE519B6B, 16#F5B95675, 16#6B58E8DA, 
		16#95AE65A3, 16#DA66BA66, 16#AA6B1AEA, 16#F601AC75, 16#4082302E, 16#8CE93226, 16#F2000AEC, 16#03C62483, 
		16#2FC18102, 16#6E076B52, 16#508B3BAD, 16#8F683131, 16#C1D66193, 16#2056FDCE;
END_VAR

(* Global variable list: LON/Module_1/Runtime_Module_1 *)
VAR_GLOBAL
(******************************************)
(* Automatic generated code, do not edit! *)
(******************************************)
	mbxModule_1 : MBX_Full;
	InDataTelegram_Module_1 : ARRAY[0..255] OF BYTE;
	OutDataTelegram_Module_1 : ARRAY[0..511] OF BYTE;

	xInitRunning_Module_1 : BOOL := FALSE;
	unLastLen_mbxModule_1 : UINT;
END_VAR

(* Data type in LON/Enumerations *)
TYPE alarm_type_t :
(
	AL_HEADER := -13,
	AL_FOOTER := -12,
	AL_DEBUG := -11,
	AL_INFO := -10,
	AL_SYSTEM_INFO := -6,
	AL_VALUE_INVALID := -5,
	AL_CONSTANT := -4,
	AL_OFFLINE := -3,
	AL_UNKNOWN := -2,
	AL_NUL := -1,
	AL_NO_CONDITION := 0,
	AL_ALM_CONDITION := 1,
	AL_TOT_SVC_ALM_1 := 2,
	AL_TOT_SVC_ALM_2 := 3,
	AL_TOT_SVC_ALM_3 := 4,
	AL_LOW_LMT_CLR_1 := 5,
	AL_LOW_LMT_CLR_2 := 6,
	AL_HIGH_LMT_CLR_1 := 7,
	AL_HIGH_LMT_CLR_2 := 8,
	AL_LOW_LMT_ALM_1 := 9,
	AL_LOW_LMT_ALM_2 := 10,
	AL_HIGH_LMT_ALM_1 := 11,
	AL_HIGH_LMT_ALM_2 := 12,
	AL_FIR_ALM := 13,
	AL_FIR_PRE_ALM := 14,
	AL_FIR_TRBL := 15,
	AL_FIR_SUPV := 16,
	AL_FIR_TEST_ALM := 17,
	AL_FIR_TEST_PRE_ALM := 18,
	AL_FIR_ENVCOMP_MAX := 19,
	AL_FIR_MONITOR_COND := 20,
	AL_FIR_MAINT_ALERT := 21,
	AL_FATAL_ERROR := 30,
	AL_ERROR := 31,
	AL_WARNING := 32
);
END_TYPE

(* Data type in Logger *)
TYPE en_Logger_ErrLev :
(
	EL_Log			:=0,
	EL_Wrn			:=1,
	EL_Alarm		:=2,
	EL_AlarmStop	:=3
);
END_TYPE

(* Data type in Logger *)
TYPE en_Logger_Status :
(
	S_Logger_UNKNOWN := 0,
	S_Logger_IDLE,
	S_Logger_WAITCONN,
	S_Logger_WAITTX,
	S_Logger_WAITRESP,
	S_Logger_ERROR
);
END_TYPE

(* Data type *)
TYPE en_SYS_Objects :
(
	EO_SYS		:=0,  (* PLC *)
	EO_VPN		:=1,  (* VPN *)
	EO_DOOR		:=2,  (* Door & access control *)

	EO_CAL		:=10, (* Caldaia *)
	EO_CIR		:=11, (* Circolatore *)
	EO_CRON		:=12, (* Crono-termostato *)
	EO_VRD		:=13, (* Valvola miscelatore pannelli *)
	EO_CTL		:=14, (* Contalitri *)
	EO_CTB		:=15, (* Contabilizzatore *)
	EO_TPV		:=16, (* Temperature probes values *)
	EO_PPV		:=17, (* Pressure probes values *)
	EO_PBV		:=18, (* Over-Pressure Alarms *)
	EO_TBV		:=19, (* Over-Temperature Alarms *)
	EO_PMV		:=20, (* Under-Pressure Alarms *)
	EO_GRU		:=21, (* Gruppo termico *)
	EO_PDC		:=22, (* Pompa di calore *)
	EO_SOL		:=23, (* Pannello solare termico *)
	EO_ESOL		:=24, (* Pannello solare fotovoltaico *)
	EO_GAS		:=25, (* Contatore GAS *)
	EO_PORT		:=26, (* Misuratore di portata *)
	EO_FPV		:=27, (* Flow probes values *)
	EO_ANZ		:=28, (* Analizzatore di rete *)
	EO_SCA		:=29, (* Signal Control Alarms *)
	EO_LUX		:=30, (* Base Illumination point *)
	EO_LUXM		:=31, (* Metered Illumination point *)
	EO_PSG		:=32, (* Sensore di passaggio *)
	EO_HVAC		:=33, (* Heating, Ventilating and Air Conditioning *)
	EO_HYGRV	:=34, (* Relative Humidity sensors value *)
	EO_COOV		:=35, (* Carbon Dioxide CO2 sensors value *)
	EO_INV		:=36, (* Inverter *)
	EO_STR		:=37, (* Smart string box *)

	EO_CIRD		:=39, (* Double CIR *)
	EO_ACS		:=40, (* Hot domestic water *)

	EO_ZGW			:=200,  (* ZigBee - Gateway *)
	EO_ZRM			:=201,	(* ZigBee - Repeater *)
	EO_ZREL			:=202,	(* ZigBee - Actuator rele *)
	EO_ZTHL			:=203,	(* ZigBee - Temperature Sensor *)

	EO_ASGW			:=250,	(* ASi - Gateway *)
	EO_ASCBI		:=251,	(* ASi - Input Board, Ciabatta *)

	EO_LON			:=1000, (* Bus - LON *)
	EO_MODBUS		:=1001, (* Bus - MODBUS *)
	EO_MBUS			:=1002, (* Bus - M-BUS *)
	EO_MODBUS_TCP	:=1003, (* Bus - MODBUS TCP *)

	EO_GENERIC		:=9000, (* Generic dataset *)
	EO_EXPO			:=9001 (* EXPO dataset *)
);
END_TYPE

(* Data type *)
TYPE en_SYS_Status :
(
	S_UNKNOWN  := 0,
	S_STARTUP,
	S_INIT_RTC,
	S_INIT_VAR,
	S_AUTOTEST,
	S_RUNNING,
	S_SHUTDOWN,
	S_HALT
);
END_TYPE

(* Data type in LON/Enumerations *)
TYPE file_request_t :
(
	FR_NUL := -1,
	FR_OPEN_TO_SEND := 0,
	FR_OPEN_TO_RECEIVE := 1,
	FR_CLOSE_FILE := 2,
	FR_CLOSE_DELETE_FILE := 3,
	FR_DIRECTORY_LOOKUP := 4,
	FR_OPEN_TO_SEND_RA := 5,
	FR_OPEN_TO_RECEIVE_RA := 6
);
END_TYPE

(* Data type in LON/Enumerations *)
TYPE file_status_t :
(
	FS_NUL := -1,
	FS_XFER_OK := 0,
	FS_LOOKUP_OK := 1,
	FS_OPEN_FAIL := 2,
	FS_LOOKUP_ERR := 3,
	FS_XFER_UNDERWAY := 4,
	FS_IO_ERR := 5,
	FS_TIMEOUT_ERR := 6,
	FS_WINDOW_ERR := 7,
	FS_AUTH_ERR := 8,
	FS_ACCESS_UNAVAIL := 9,
	FS_SEEK_INVALID := 10,
	FS_SEEK_WAIT := 11
);
END_TYPE

(* Data type in LON/Enumerations *)
TYPE hvac_t :
(
	HVAC_NUL := -1,
	HVAC_AUTO := 0,
	HVAC_HEAT := 1,
	HVAC_MRNG_WRMUP := 2,
	HVAC_COOL := 3,
	HVAC_NIGHT_PURGE := 4,
	HVAC_PRE_COOL := 5,
	HVAC_OFF := 6,
	HVAC_TEST := 7,
	HVAC_EMERG_HEAT := 8,
	HVAC_FAN_ONLY := 9,
	HVAC_FREE_COOL := 10,
	HVAC_ICE := 11,
	HVAC_MAX_HEAT := 12,
	HVAC_ECONOMY := 13,
	HVAC_DEHUMID := 14,
	HVAC_CALIBRATE := 15,
	HVAC_EMERG_COOL := 16,
	HVAC_EMERG_STEAM := 17,
	HVAC_MAX_COOL := 18,
	HVAC_HVC_LOAD := 19,
	HVAC_NO_LOAD := 20
);
END_TYPE

(* Data type in LON/Enumerations *)
TYPE object_request_t :
(
	RQ_NUL := -1,
	RQ_NORMAL := 0,
	RQ_DISABLED := 1,
	RQ_UPDATE_STATUS := 2,
	RQ_SELF_TEST := 3,
	RQ_UPDATE_ALARM := 4,
	RQ_REPORT_MASK := 5,
	RQ_OVERRIDE := 6,
	RQ_ENABLE := 7,
	RQ_RMV_OVERRIDE := 8,
	RQ_CLEAR_STATUS := 9,
	RQ_CLEAR_ALARM := 10,
	RQ_ALARM_NOTIFY_ENABLED := 11,
	RQ_ALARM_NOTIFY_DISABLED := 12,
	RQ_MANUAL_CTRL := 13,
	RQ_REMOTE_CTRL := 14,
	RQ_PROGRAM := 15,
	RQ_CLEAR_RESET := 16,
	RQ_RESET := 17,
	RQ_CLEAR_LOG := 18,
	RQ_LOAD_PROGRAM := 19,
	RQ_RUN_PROGRAM := 20,
	RQ_HALT_PROGRAM := 21,
	RQ_RESTART_PROGRAM := 22,
	RQ_UNLOAD_PROGRAM := 23,
	RQ_STEP_PROGRAM := 24
);
END_TYPE

(* Data type in LON/Enumerations *)
TYPE priority_level_t :
(
	PR_NUL := -1,
	PR_LEVEL_0 := 0,
	PR_LEVEL_1 := 1,
	PR_LEVEL_2 := 2,
	PR_LEVEL_3 := 3,
	PR_1 := 4,
	PR_2 := 5,
	PR_3 := 6,
	PR_4 := 7,
	PR_6 := 8,
	PR_8 := 9,
	PR_10 := 10,
	PR_16 := 11
);
END_TYPE

(* Data type in Plant_Objects *)
TYPE typ_Clima : (* CURVA CLIMATICA *)
STRUCT
	InitOK:		BOOL;
	Points: 	ARRAY [0..10] OF POINT;
END_STRUCT
END_TYPE

(* Data type in Plant_Objects *)
TYPE typ_Cron_Calendar :
STRUCT
	Profile		: ARRAY[0..384] OF BYTE;
END_STRUCT
END_TYPE

(* Data type in Plant_Objects *)
TYPE typ_Cron_Jolly :
STRUCT
	Start		: DT;
	End			: DT;
	Temp		: WORD;
	Flags		: WORD; (* B0:Enabled B1..B15:Unused *)
END_STRUCT
END_TYPE

(* Data type in Plant_Objects *)
TYPE typ_Cron_Profile :
STRUCT
	Flags		: WORD;
	Setpoint	: ARRAY [0..95] OF WORD;
END_STRUCT
END_TYPE

(* Data type in Plant_Objects *)
TYPE typ_Frigo :
STRUCT
	Status	:	BOOL;		(* 0=OFF, 1=ON	*)
	Mode	:	BOOL;		(* 0=COLD, 1=HOT	*)

END_STRUCT
END_TYPE

(* Data type in Logger *)
TYPE typ_Logger :
STRUCT
	Status		: en_Logger_Status;

	SendReq		: BOOL;
	SendIdx		: DWORD;
	SendData	: ARRAY [0..MAX_SEND_TCP_CLIENT] OF BYTE;
	SendLen		: DINT;

	TData		: ARRAY [0..MAX_SEND_TCP_CLIENT] OF BYTE;
	TLen		: DINT;

	LastIdxPos	: DWORD;

	(* Temporary variables used by objects *)
	s1			: STRING(256);
	i1			: WORD;

END_STRUCT
END_TYPE

(* Data type in Plant_Objects *)
TYPE typ_MODBUS_CIR :
STRUCT
	PumpStatus		:	WORD;
	PumpFault		:	BOOL;
	PumpBoardTemp	:	INT;	(* Electonic board temperature  [°C] *)
	PumpVoltage		:	WORD;	(* Input voltage rms [V] *)
	PumpCurrent		:	WORD;	(* Output current [E-3 A]	*)
	PumpRPM			:	WORD;	(* Round per minute [rpm] *)
	PumpPower		:	WORD;	(* Power [W] *)
	PumpOpTime		:	DWORD;	(* Pump operating time [h] *)
	PumpHead		:	WORD;	(* [E-1 m] *)
	PumpFlow		:	WORD;	(* Extimated flow [E-1 m3/h] *)
	PumpLiqTemp		:	WORD;	(* Liquid temperature [°C] *)
	PumpAlarm		:	ARRAY [0..14] OF WORD;

END_STRUCT
END_TYPE

(* Data type in Plant_Objects *)
TYPE typ_MODBUS_VAR : (* Gestione parametri MODBUS *)
STRUCT
	SlaveAddress	: BYTE;
	FunCode			: BYTE;
	FunAddress		: WORD;
	Refresh_Time	: BYTE; (* 0:No refresh x:Refresh in seconds *)
	Refresh_Cnt		: BYTE; (* INTERNAL *)
	Variable		: POINTER TO WORD;
	Variable_Size	: BYTE;
	Variable_Mirror : WORD; (* INTERNAL [Force refresh on read variables when <>0] *)
END_STRUCT
END_TYPE

(* Data type *)
TYPE typ_SYS :
STRUCT
	Status			: en_SYS_Status;
	Warning			: BOOL;
	Alarm			: BOOL;
	AlarmStop		: BOOL;

	Time_LogString	: STRING;
	Time_Year		: WORD;
	Time_Month		: BYTE;
	Time_Day		: BYTE;

	Time_CT_DT		: DT;
	Time_CT_Day		: WORD;
	Time_CT_Quarter	: BYTE;

	LastLogs_Idx	: BYTE;
	LastLogs_Dat	: ARRAY[0..5] OF STRING;
	LastLogs_Msg	: ARRAY[0..5] OF STRING;

END_STRUCT
END_TYPE

(* Data type in Plant_Objects *)
TYPE typ_VisuStrutturaMbus :
STRUCT

	sdNodoPresente: STRING(16);
	sdEnergia: STRING(16);
	sdPotenza: STRING(16);
	sdVolume: STRING(16);
	sdFlow: STRING(16);
	sdTempIngresso: STRING(8);
	sdTempaUscita: STRING(8);
	sdTempDelta: STRING(8);

END_STRUCT
END_TYPE

(* Data type in LON/NetworkVariables *)
TYPE typSnvtAlarm : 
STRUCT
	abLocation : ARRAY[0..5] OF BYTE;
	wObjectId : WORD;
	bAlarmType : BYTE (* enum type alarm_type_t *);
	bPriorityLevel : BYTE (* enum type priority_level_t *);
	wIndexToSnvt : WORD;
	abValue : ARRAY[0..3] OF BYTE;
	wYear : WORD;
	bMonth : BYTE;
	bDay : BYTE;
	bHour : BYTE;
	bMinute : BYTE;
	bSecond : BYTE;
	wMillisecond : WORD;
	abAlarmLimit : ARRAY[0..3] OF BYTE;
	bStatusInformation : BYTE; (* bit allocation of bStatusInformation:
	bit 0: NVI update counter LSB
	bit 1: NVI update counter
	bit 2: NVI update counter
	bit 3: NVI update counter MSB
	bit 4: timeout for NVI occurs (MaxRcvTime expired)
	bit 5: reserved
	bit 6: reserved
	bit 7: force NVO update *)
	bInternalUseOnly : BYTE; (* Do not use this byte in your application! *)
END_STRUCT
END_TYPE

(* Data type in LON/NetworkVariables *)
TYPE typSnvtFilePos : 
STRUCT
	diRwPtr : DINT;
	wRwLength : WORD;
	bStatusInformation : BYTE; (* bit allocation of bStatusInformation:
	bit 0: NVI update counter LSB
	bit 1: NVI update counter
	bit 2: NVI update counter
	bit 3: NVI update counter MSB
	bit 4: timeout for NVI occurs (MaxRcvTime expired)
	bit 5: reserved
	bit 6: reserved
	bit 7: force NVO update *)
	bInternalUseOnly : BYTE; (* Do not use this byte in your application! *)
END_STRUCT
END_TYPE

(* Data type in LON/NetworkVariables *)
TYPE typSnvtFileReq : 
STRUCT
	bRequest : BYTE (* enum type file_request_t *);
	wIndex : WORD;
	wReceiveTimeout : WORD;
	abDestAddress : ARRAY[0..4] OF BYTE (* union declaration *);
	bAuthOn : BYTE;
	bPrioOn : BYTE;
	bStatusInformation : BYTE; (* bit allocation of bStatusInformation:
	bit 0: NVI update counter LSB
	bit 1: NVI update counter
	bit 2: NVI update counter
	bit 3: NVI update counter MSB
	bit 4: timeout for NVI occurs (MaxRcvTime expired)
	bit 5: reserved
	bit 6: reserved
	bit 7: force NVO update *)
	bInternalUseOnly : BYTE; (* Do not use this byte in your application! *)
END_STRUCT
END_TYPE

(* Data type in LON/NetworkVariables *)
TYPE typSnvtFileStatus : 
STRUCT
	bStatus : BYTE (* enum type file_status_t *);
	wNumberOfFiles : WORD;
	wSelectedFile : WORD;
	abAdr : ARRAY[0..21] OF BYTE (* union declaration *);
	bStatusInformation : BYTE; (* bit allocation of bStatusInformation:
	bit 0: NVI update counter LSB
	bit 1: NVI update counter
	bit 2: NVI update counter
	bit 3: NVI update counter MSB
	bit 4: timeout for NVI occurs (MaxRcvTime expired)
	bit 5: reserved
	bit 6: reserved
	bit 7: force NVO update *)
	bInternalUseOnly : BYTE; (* Do not use this byte in your application! *)
END_STRUCT
END_TYPE

(* Data type in LON/NetworkVariables *)
TYPE typSnvtHvacMode : 
STRUCT
	bSnvtHvacMode : BYTE (* enum type hvac_t *);
	bStatusInformation : BYTE; (* bit allocation of bStatusInformation:
	bit 0: NVI update counter LSB
	bit 1: NVI update counter
	bit 2: NVI update counter
	bit 3: NVI update counter MSB
	bit 4: timeout for NVI occurs (MaxRcvTime expired)
	bit 5: reserved
	bit 6: reserved
	bit 7: force NVO update *)
	bInternalUseOnly : BYTE; (* Do not use this byte in your application! *)
END_STRUCT
END_TYPE

(* Data type in LON/NetworkVariables *)
TYPE typSnvtObjRequest : 
STRUCT
	wObjectId : WORD;
	bObjectRequest : BYTE (* enum type object_request_t *);
	bStatusInformation : BYTE; (* bit allocation of bStatusInformation:
	bit 0: NVI update counter LSB
	bit 1: NVI update counter
	bit 2: NVI update counter
	bit 3: NVI update counter MSB
	bit 4: timeout for NVI occurs (MaxRcvTime expired)
	bit 5: reserved
	bit 6: reserved
	bit 7: force NVO update *)
	bInternalUseOnly : BYTE; (* Do not use this byte in your application! *)
END_STRUCT
END_TYPE

(* Data type in LON/NetworkVariables *)
TYPE typSnvtObjStatus : 
STRUCT
	wObjectId : WORD;
	bBitfieldByteOffset2 : BYTE (* bit field *);
	bBitfieldByteOffset3 : BYTE (* bit field *);
	bBitfieldByteOffset4 : BYTE (* bit field *);
	bBitfieldByteOffset5 : BYTE (* bit field *);
	bStatusInformation : BYTE; (* bit allocation of bStatusInformation:
	bit 0: NVI update counter LSB
	bit 1: NVI update counter
	bit 2: NVI update counter
	bit 3: NVI update counter MSB
	bit 4: timeout for NVI occurs (MaxRcvTime expired)
	bit 5: reserved
	bit 6: reserved
	bit 7: force NVO update *)
	bInternalUseOnly : BYTE; (* Do not use this byte in your application! *)
END_STRUCT
END_TYPE

(* Data type in LON/NetworkVariables *)
TYPE typSnvtState : 
STRUCT
	bBitfieldByteOffset0 : BYTE (* bit field *);
	bBitfieldByteOffset1 : BYTE (* bit field *);
	bStatusInformation : BYTE; (* bit allocation of bStatusInformation:
	bit 0: NVI update counter LSB
	bit 1: NVI update counter
	bit 2: NVI update counter
	bit 3: NVI update counter MSB
	bit 4: timeout for NVI occurs (MaxRcvTime expired)
	bit 5: reserved
	bit 6: reserved
	bit 7: force NVO update *)
	bInternalUseOnly : BYTE; (* Do not use this byte in your application! *)
END_STRUCT
END_TYPE

(* Data type in LON/NetworkVariables *)
TYPE typSnvtSwitch : 
STRUCT
	bValue : BYTE;
	siState : SINT;
	bStatusInformation : BYTE; (* bit allocation of bStatusInformation:
	bit 0: NVI update counter LSB
	bit 1: NVI update counter
	bit 2: NVI update counter
	bit 3: NVI update counter MSB
	bit 4: timeout for NVI occurs (MaxRcvTime expired)
	bit 5: reserved
	bit 6: reserved
	bit 7: force NVO update *)
	bInternalUseOnly : BYTE; (* Do not use this byte in your application! *)
END_STRUCT
END_TYPE

(* Data type in LON/NetworkVariables *)
TYPE typSnvtTempP : 
STRUCT
	iSnvtTempP : INT;
	bStatusInformation : BYTE; (* bit allocation of bStatusInformation:
	bit 0: NVI update counter LSB
	bit 1: NVI update counter
	bit 2: NVI update counter
	bit 3: NVI update counter MSB
	bit 4: timeout for NVI occurs (MaxRcvTime expired)
	bit 5: reserved
	bit 6: reserved
	bit 7: force NVO update *)
	bInternalUseOnly : BYTE; (* Do not use this byte in your application! *)
END_STRUCT
END_TYPE

(* Data type in LON/NetworkVariables *)
TYPE typSnvtTimeStamp : 
STRUCT
	iYear : INT;
	bMonth : BYTE;
	bDay : BYTE;
	bHour : BYTE;
	bMinute : BYTE;
	bSecond : BYTE;
	bStatusInformation : BYTE; (* bit allocation of bStatusInformation:
	bit 0: NVI update counter LSB
	bit 1: NVI update counter
	bit 2: NVI update counter
	bit 3: NVI update counter MSB
	bit 4: timeout for NVI occurs (MaxRcvTime expired)
	bit 5: reserved
	bit 6: reserved
	bit 7: force NVO update *)
	bInternalUseOnly : BYTE; (* Do not use this byte in your application! *)
END_STRUCT
END_TYPE

(* POU PLC_PRG, ST *)
PROGRAM PLC_PRG
VAR
	Timer1: TON; (* Fast controls tick *)
	Timer2: TON; (* Plant control tick *)
	Timer3: TON; (* Logger timer *)

	T_CIR01		:	INT;
	T_CIR02		:	INT;
	T_CIR03		:	INT;
	T_CIR04		:	INT;
	T_CIRD01	:	INT;

	T_Valve01	:	INT;
	T_Valve02	:	INT;
	T_Valve03	:	INT;

END_VAR
(******************************************************************************
 ****                           MAIN TASK CODE                             ****
 ******************************************************************************

	Network setup:
		IP  = 192.168.100.2 | MSK = 255.255.255.0
		GW	= 192.168.100.1 | DNS = 192.168.100.1
		SNTP = 193.204.114.232 (3600s) ==> 192.168.100.3

*)

(*==============================*)
(*===== Main status machine ====*)
(*==============================*)
Main_Stm();

(*==============================*)
(*== Running cycle operations ==*)
(*==============================*)
IF SYS.Status>S_INIT_VAR THEN
	(* Execute cycle processes *)
	(* Update LON output variables (needs to be here to obtain only one refresh) *)
	GRU01.Heartbeat( CLIM:=GRU01_Clima );

	(* Execute LON process *)
	Module_1_PRG();

	(* Count water pulses *)
	CTL01(CTL_ST:=CTL01_ST, COUNT:=Ctl01_Counter);

	(* ModBus *)
	MODB01();

	CIR02(ModBus:=MODB01, CIR_AL:=NOT CIR02_AL, CIR_AUTO:=CIR02_AUTO);
	CIR03(ModBus:=MODB01, CIR_AL:=NOT CIR03_AL, CIR_AUTO:=CIR03_AUTO);

	CIRD01(ModBus:=MODB01, PumpA_AL:=NOT CIRD01_A_AL, PumpB_AL:=NOT CIRD01_B_AL, PumpA_AUTO:=CIRD01_A_AUTO, PumpB_AUTO:=CIRD01_B_AUTO);

	(* M-Bus *)
	MBUS01();

	CTB01(MBUS:=MBUS01);
	CTB02(MBUS:=MBUS01);

END_IF

(*==============================*)
(*== System cycle operations ===*)
(*==============================*)
(* Execute TCP processes *)
Logger_Proc();
Remote_Proc();
(* Update user led *)
USRLED_Update();
(* Execute Cron Editor commands *)
CronEd();

(* Environment temperature *)
IF NOT TPV01.ERR THEN T_AMB := S01;
ELSE T_AMB := Plant_DefaultTAmb;
END_IF


(**** SIMULATION ONLY ****)
(*...*)
END_PROGRAM
ACTION Main_Stm:
CASE Sys.Status OF

	S_STARTUP:
		Sys.Status:=S_INIT_RTC;

	S_INIT_RTC:
		(* Check RTC and update from network *)
		RTC_Update();
		(* Check time *)
		IF Sys.Time_Year>2000 THEN
			Sys.Status:=S_INIT_VAR;
		END_IF

	S_INIT_VAR:
		LogEv(EL_Wrn,EO_SYS,0,1,CONCAT('System_startup_v',WORD_TO_STRING(Plant_SW_VER)));
		Sys.Status:=S_RUNNING;

	S_RUNNING:
		Timer1(IN:=NOT Timer1.Q,PT:=T#50ms);
		IF Timer1.Q THEN
			(* Update meters *)

			(* Update system checks *)
			SYS_Proc();
		END_IF

		Timer2(IN:=NOT Timer2.Q,PT:=T#500ms);
		IF Timer2.Q THEN
			(* Read current date/time *)
			RTC_Update();

			(* Boiler *)

			(* Probes *)
			TPV01();
			TPV02();
			TPV03();
			TPV04();
			TPV05();
			TPV06();
			TPV07();
			TPV08();
			TPV09();
			TPV10();
			TPV11();
			TPV12();

			(* Temperature *)
			TPV02.Mean();
			T_CIR02 := SEL(TPV02.ERR,TPV02.AVG,450);

			TPV08.Mean();
			T_CIR04 := SEL(TPV08.ERR,TPV08.AVG,Plant_DefaultTAmb);

			TPV09.Mean();
			T_CIR03 := SEL(TPV09.ERR,TPV09.AVG,Plant_DefaultTAmb);

			TPV10.Mean();
			TPV11.Mean();
			TPV12.Mean();
			T_CIRD01 := MUX_T(T1:=TPV10.AVG, T2:=TPV11.AVG, T3:=TPV12.AVG,
							  Err1:=TPV10.ERR, Err2:=TPV11.ERR, Err3:=TPV12.ERR, Used:=3);

			TPV05.Mean();
			T_Valve01 := SEL(TPV05.ERR,TPV05.AVG,Plant_VRD_TDefault);
			TPV06.Mean();
			T_Valve02 := SEL(TPV06.ERR,TPV06.AVG,Plant_VRD_TDefault);
			TPV04.Mean();
			T_Valve03 := SEL(TPV04.ERR,TPV04.AVG,Plant_VRD_TDefault);

			(* Thermostats *)
			THER01(Temperature:=T_CIR03, Run=>CIR03.OnOff);
			THER02(Temperature:=T_CIR04, Run=>CIR04.OnOff);
			THER03(Temperature:=T_CIRD01, Run=>CIRD01.OnOff);
			THER04(Temperature:=T_CIR02, Run=>CIR02.OnOff);

			(*Hot domestic water *)
			ACS01();

			(* CAL *)
			CAL04(OnOff:=BYTE_TO_BOOL(ACS01.Run), Alarm:=CAL01_AL, Status:=CAL01_ST, Enable=>CAL01_EN, Reset=>CAL01_RST);

			(* CIR *)
			CIR04(CIR_AL:=NOT CIR04_AL, CIR_ST:=CIR04_ST, CIR_AUTO:=CIR04_AUTO);
			(* Cir01 is related to CIR04 working *)
			CIR01(OnOff:=BOOL_TO_BYTE(CIR04.Run), CIR_AL:=NOT CIR01_AL, CIR_ST:=CIR01_ST, CIR_AUTO:=CIR01_AUTO);

			(* Valves *)
			VRD01(RUN:=CIR03.Run, CLIM:=VRD01_Clima, TEMP:=T_Valve01, STATUS:=VRD01_ST, OUT=>VRD01_CTRL);
			VRD02(RUN:=CIR04.Run, CLIM:=VRD02_Clima, TEMP:=T_Valve02, STATUS:=VRD02_ST, OUT=>VRD02_CTRL);
			VRD03(RUN:=CIRD01.Run, CLIM:=VRD03_Clima, TEMP:=T_Valve03, STATUS:=VRD03_ST, OUT=>VRD03_CTRL);

			(* Check plant status *)
			Lamp();

			(* Test toggle *)
			(*IF TEST1 THEN TEST1:=FALSE; ELSE TEST1:=TRUE; END_IF*)
		END_IF

		Timer3(IN:=NOT Timer3.Q,PT:=T#5m);
		IF Timer3.Q THEN
			(* Trig logger *)
			LogTrig();
			(* Execute temporary CSV logger *)
			(*CSV_Log();*)
		END_IF

	S_SHUTDOWN:
		(* Stop sistema *)
		Sys.Status:=S_STARTUP;

	S_HALT:
		(* Aspetta uscita manuale *)
		Sys.Status:=S_STARTUP;

ELSE
	Sys.Status:=S_STARTUP;
END_CASE;
END_ACTION

(* POU LON/Module_1/Module_1_PRG, FBD *)
PROGRAM Module_1_PRG
VAR
	(* Automatic added code, do not change! *)
	LonMaster : Module_1_LonMaster;
	SFPTnodeObject : Module_1_SFPTnodeObject;
	Virtualfunctionalblock : Module_1_Virtualfunctionalblock;

	InData_LON AT %IB24 : ARRAY[0..23] OF BYTE;
	OutData_LON AT %QB0 : ARRAY[0..23] OF BYTE;
	(***** End of automatic added code. *****)

	(* Add your code here. *)

	LonState: BOOL;
	LonReset: BOOL;
END_VAR
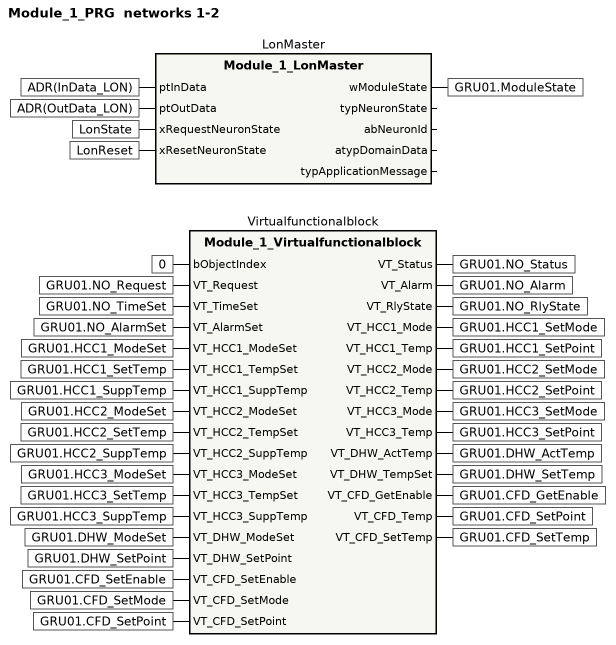
_FBD_ (* Function Block Diagram *)
NETWORK 1 (* Added by code generator *)
	LonMaster:Module_1_LonMaster(ptInData: ADR(InData_LON), ptOutData: ADR(OutData_LON), xRequestNeuronState: LonState, xResetNeuronState: LonReset) => GRU01.ModuleState
NETWORK 2
	Virtualfunctionalblock:Module_1_Virtualfunctionalblock(bObjectIndex: 0, VT_Request: GRU01.NO_Request, VT_TimeSet: GRU01.NO_TimeSet, VT_AlarmSet: GRU01.NO_AlarmSet, VT_HCC1_ModeSet: GRU01.HCC1_ModeSet, VT_HCC1_TempSet: GRU01.HCC1_SetTemp, VT_HCC1_SuppTemp: GRU01.HCC1_SuppTemp, VT_HCC2_ModeSet: GRU01.HCC2_ModeSet, VT_HCC2_TempSet: GRU01.HCC2_SetTemp, VT_HCC2_SuppTemp: GRU01.HCC2_SuppTemp, VT_HCC3_ModeSet: GRU01.HCC3_ModeSet, VT_HCC3_TempSet: GRU01.HCC3_SetTemp, VT_HCC3_SuppTemp: GRU01.HCC3_SuppTemp, VT_DHW_ModeSet: GRU01.DHW_ModeSet, VT_DHW_SetPoint: GRU01.DHW_SetPoint, VT_CFD_SetEnable: GRU01.CFD_SetEnable, VT_CFD_SetMode: GRU01.CFD_SetMode, VT_CFD_SetPoint: GRU01.CFD_SetPoint, VT_Alarm => GRU01.NO_Alarm, VT_RlyState => GRU01.NO_RlyState, VT_HCC1_Mode => GRU01.HCC1_SetMode, VT_HCC1_Temp => GRU01.HCC1_SetPoint, VT_HCC2_Mode => GRU01.HCC2_SetMode, VT_HCC2_Temp => GRU01.HCC2_SetPoint, VT_HCC3_Mode => GRU01.HCC3_SetMode, VT_HCC3_Temp => GRU01.HCC3_SetPoint, VT_DHW_ActTemp => GRU01.DHW_ActTemp, VT_DHW_TempSet => GRU01.DHW_SetTemp, VT_CFD_GetEnable => GRU01.CFD_GetEnable, VT_CFD_Temp => GRU01.CFD_SetPoint, VT_CFD_SetTemp => GRU01.CFD_SetTemp) => GRU01.NO_Status
_END_FBD_
(* the same logic as Structured Text *)
(* Network 1: Added by code generator *)
LonMaster(ptInData := ADR(InData_LON), ptOutData := ADR(OutData_LON), xRequestNeuronState := LonState, xResetNeuronState := LonReset);
GRU01.ModuleState := LonMaster.wModuleState;
(* Network 2 *)
Virtualfunctionalblock(bObjectIndex := 0, VT_Request := GRU01.NO_Request, VT_TimeSet := GRU01.NO_TimeSet, VT_AlarmSet := GRU01.NO_AlarmSet, VT_HCC1_ModeSet := GRU01.HCC1_ModeSet, VT_HCC1_TempSet := GRU01.HCC1_SetTemp, VT_HCC1_SuppTemp := GRU01.HCC1_SuppTemp, VT_HCC2_ModeSet := GRU01.HCC2_ModeSet, VT_HCC2_TempSet := GRU01.HCC2_SetTemp, VT_HCC2_SuppTemp := GRU01.HCC2_SuppTemp, VT_HCC3_ModeSet := GRU01.HCC3_ModeSet, VT_HCC3_TempSet := GRU01.HCC3_SetTemp, VT_HCC3_SuppTemp := GRU01.HCC3_SuppTemp, VT_DHW_ModeSet := GRU01.DHW_ModeSet, VT_DHW_SetPoint := GRU01.DHW_SetPoint, VT_CFD_SetEnable := GRU01.CFD_SetEnable, VT_CFD_SetMode := GRU01.CFD_SetMode, VT_CFD_SetPoint := GRU01.CFD_SetPoint);
GRU01.NO_Alarm := Virtualfunctionalblock.VT_Alarm;
GRU01.NO_RlyState := Virtualfunctionalblock.VT_RlyState;
GRU01.HCC1_SetMode := Virtualfunctionalblock.VT_HCC1_Mode;
GRU01.HCC1_SetPoint := Virtualfunctionalblock.VT_HCC1_Temp;
GRU01.HCC2_SetMode := Virtualfunctionalblock.VT_HCC2_Mode;
GRU01.HCC2_SetPoint := Virtualfunctionalblock.VT_HCC2_Temp;
GRU01.HCC3_SetMode := Virtualfunctionalblock.VT_HCC3_Mode;
GRU01.HCC3_SetPoint := Virtualfunctionalblock.VT_HCC3_Temp;
GRU01.DHW_ActTemp := Virtualfunctionalblock.VT_DHW_ActTemp;
GRU01.DHW_SetTemp := Virtualfunctionalblock.VT_DHW_TempSet;
GRU01.CFD_GetEnable := Virtualfunctionalblock.VT_CFD_GetEnable;
GRU01.CFD_SetPoint := Virtualfunctionalblock.VT_CFD_Temp;
GRU01.CFD_SetTemp := Virtualfunctionalblock.VT_CFD_SetTemp;
GRU01.NO_Status := Virtualfunctionalblock.VT_Status;
END_PROGRAM

(* POU LON/Module_1/Master/Module_1_LonMaster, ST *)
FUNCTION_BLOCK Module_1_LonMaster
(******************************************)
(* Automatic generated code, do not edit! *)
(******************************************)
VAR_INPUT
	ptInData  : POINTER TO BYTE;
	ptOutData : POINTER TO BYTE;
	xRequestNeuronState : BOOL;
	xResetNeuronState : BOOL;
END_VAR
VAR_OUTPUT
	wModuleState : WORD; (* bit coded wModuleState:
	15: communication to I/O-module interrupted (error)
	14 - 08: reserved
	07: ready for Neuron initialization
	06: Neuron active
	05: user interface active
	04: internal module communication interrupted (error)
	03: CP synchronization running
	02: Neuron is configured online
	01 - 00: reserved *)

	typNeuronState : NeuronState;
	abNeuronId : ARRAY[0..5] OF BYTE;
	atypDomainData : ARRAY[0..1] OF DomainData;
	typApplicationMessage : ApplicationMessageData;
END_VAR
VAR
	bInternalCode : BYTE;
	bNvIndex : BYTE;
	wCpIndex : WORD;
	lonCom : FbLonBasicCommunication;

	xInitIsStarted : BOOL := FALSE;

	TimeoutTimer : TON;
	timeOutTime : TIME := T#1000ms;
	xStateMachineIsChecked : BOOL;
	xTimerStart : BOOL;

	iDomainTable : INT;
	xSendRequestPending : BOOL;
	trigRequest : R_TRIG;
	trigReset : R_TRIG;

	abMbxRxPrio0Buf: ARRAY [0..309] OF BYTE;
	abMbxRxPrio1Buf: ARRAY [0..517] OF BYTE;
	aMbxRxBufSize: ARRAY [0..1] OF UINT := 310, 518;
	aMbxRxBufList: ARRAY [0..1] OF POINTER TO BYTE;
	afbMbxRxFb: ARRAY [0..1] OF MBX2_RX_DEFRAG;
	astMbxRxCtx: ARRAY [0..1] OF stMbx2DefragContext;

	abMbxTxPrio0Buf: ARRAY [0..309] OF BYTE;
	abMbxTxPrio1Buf: ARRAY [0..517] OF BYTE;
	aMbxTxBufSize: ARRAY [0..1] OF UINT := 310, 518;
	aMbxTxBufList: ARRAY [0..1] OF POINTER TO BYTE;
	afbMbxTxFb: ARRAY [0..1] OF MBX2_TX_FRAG;

	astMbxTrackContext: ARRAY [0..0] OF stMbx2TrackContext;
END_VAR
VAR CONSTANT
END_VAR
aMbxRxBufList[0] := ADR(abMbxRxPrio0Buf[0]);
aMbxRxBufList[1] := ADR(abMbxRxPrio1Buf[0]);

aMbxTxBufList[0] := ADR(abMbxTxPrio0Buf[0]);
aMbxTxBufList[1] := ADR(abMbxTxPrio1Buf[0]);

mbxModule_1.Ressources.pDefragBufList := ADR(aMbxRxBufList);
mbxModule_1.Ressources.pDefragBufSizeList := ADR(aMbxRxBufSize);
mbxModule_1.Ressources.pDefragCtxPtrList := ADR(astMbxRxCtx);
mbxModule_1.Ressources.pDefragFbList := ADR(afbMbxRxFb);
mbxModule_1.Ressources.pFragBufList := ADR(aMbxTxBufList);
mbxModule_1.Ressources.pFragBufSizeList := ADR(aMbxTxBufSize);
mbxModule_1.Ressources.pFragFbList := ADR(afbMbxTxFb);

mbxModule_1.Ressources.unMaxAvailableRxPrioIndex := 1;
mbxModule_1.Ressources.unMaxAvailableTxPrioIndex := 1;

mbxModule_1.Ressources.pTrackStList := ADR(astMbxTrackContext);
mbxModule_1.Ressources.unMaxAvailableTrackIndex := 0;

mbxModule_1.Ressources.pabRxWin := ptInData + 1;
mbxModule_1.Ressources.pabTxWin := ptOutData + 1;
mbxModule_1.Ressources.bTxWinSize := 23;
mbxModule_1.Ressources.bRxWinSize := 23;

IF (mbxModule_1.bStatus.2 = TRUE) OR (mbxModule_1.bStatus.1 = TRUE) THEN
	mbxModule_1.MBX_RESET();
	xInitRunning_Module_1 := TRUE;
	xInitIsStarted := FALSE;
END_IF
mbxModule_1.MBX_CYCLE();

IF (mbxModule_1.bStatus.0 <> TRUE) THEN 
	wModuleState := 16#8000;
	RETURN;
ELSE
	wModuleState.15 := FALSE;
END_IF

xStateMachineIsChecked := FALSE;
IF xInitRunning_Module_1 = TRUE THEN
	IF xInitIsStarted = FALSE THEN
		SetParameter();
		lonCom.eInitState := INIT_SND_SGNTR_REQ;
		lonCom.CheckInitState();
		xInitIsStarted := TRUE;
		xStateMachineIsChecked := TRUE;
	END_IF
END_IF

typApplicationMessage.xMsgRcvd := FALSE;
typApplicationMessage.xRspRcvd := FALSE;
ResetNviUpdate();
WHILE (mbxModule_1.xRxPending) DO
	unLastLen_mbxModule_1 := mbxModule_1.unRxLen;
	mbxModule_1.pbRxData := ADR(InDataTelegram_Module_1);
	mbxModule_1.MBX_RETRIEVE();
	IF (mbxModule_1.nError <> MBX_OK) THEN EXIT; END_IF;
	bInternalCode := InDataTelegram_Module_1[0];

	IF (xInitRunning_Module_1 = TRUE) AND (lonCom.eInitState <> INIT_TRANSFER_CFG) THEN
		IF (FuCheckForValidInitCode(bInternalCode)) THEN
			SetParameter();
			lonCom.unLastLen := unLastLen_mbxModule_1;
			lonCom.CheckInitState();
			xInitRunning_Module_1 := NOT lonCom.xInitDone;
			xStateMachineIsChecked := TRUE;
		END_IF
	END_IF

	IF (bInternalCode = M2C_NVI_UPDT_OCCD) OR (bInternalCode = M2C_NV_VALUE_RSP) OR (bInternalCode = M2C_NVI_UPDT_TOUT) THEN
		bNvIndex := InDataTelegram_Module_1[1];
		CASE bNvIndex OF
			0, 2, 4: Module_1_PRG.SFPTnodeObject.DataReceived();
			6, 8, 10, 12, 14, 17, 19, 22, 24, 27, 29, 31, 33, 35: Module_1_PRG.Virtualfunctionalblock.DataReceived();

		END_CASE;
	ELSIF (bInternalCode = M2C_CP_VALUE_RSP) THEN
		wCpIndex := InDataTelegram_Module_1[1] OR (InDataTelegram_Module_1[2] * 256);
		CASE wCpIndex OF

		END_CASE;
	ELSIF (bInternalCode = M2C_LON_MSG_RCVD) OR (bInternalCode = M2C_LON_RSP_RCVD) THEN
		ApplMsgReceived();
	ELSIF (bInternalCode = M2C_STATUS_RSP) THEN
		wModuleState := (wModuleState AND 16#FF00) + InDataTelegram_Module_1[1];
	ELSIF (bInternalCode = M2C_NEURON_ID) THEN
		FuMemCopy(ADR(InDataTelegram_Module_1[1]), ADR(abNeuronId), 6);
	ELSIF (bInternalCode = M2C_DOMAIN_DATA) THEN
		DomainDataRcvd();
	ELSIF (bInternalCode = M2C_MICRO_SERVER_STATUS_RSP) THEN
		NeuronStateRcvd();
	END_IF
END_WHILE

IF (xInitRunning_Module_1 = TRUE) AND ((lonCom.xCallStateMachine = TRUE) OR (TimeoutTimer.Q = TRUE)) AND (NOT xStateMachineIsChecked) THEN
	SetParameter();
	lonCom.xTimeOut := TimeoutTimer.Q;
	lonCom.CheckInitState();
END_IF
TimeoutTimer(IN:=lonCom.xTimerStart, PT:=timeOutTime);

trigRequest(CLK := xRequestNeuronState);
trigReset(CLK := xResetNeuronState);
IF (trigRequest.Q OR trigReset.Q) THEN
	RequestNeuronState();
END_IF
END_FUNCTION_BLOCK
ACTION ApplMsgReceived:
IF (InDataTelegram_Module_1[0] = M2C_LON_MSG_RCVD) THEN
	typApplicationMessage.typService := InDataTelegram_Module_1[1] AND 16#30;
	typApplicationMessage.bSourceSubnetId := InDataTelegram_Module_1[2];
	typApplicationMessage.bSourceNodeId := InDataTelegram_Module_1[3];
	typApplicationMessage.bCorrelator := InDataTelegram_Module_1[4];
	typApplicationMessage.bCode :=  InDataTelegram_Module_1[5];
	typApplicationMessage.bDataLength := UINT_TO_BYTE(unLastLen_mbxModule_1 - 6);
	IF typApplicationMessage.bDataLength > 48 THEN typApplicationMessage.bDataLength := 48; END_IF;
	FuMemSet(ADR(typApplicationMessage.abData), 0, SIZEOF(typApplicationMessage.abData));
	IF typApplicationMessage.bDataLength > 0 THEN
		FuMemCopy(ADR(InDataTelegram_Module_1[6]), ADR(typApplicationMessage.abData), typApplicationMessage.bDataLength);
	END_IF
	typApplicationMessage.xMsgRcvd := TRUE;
ELSE
	typApplicationMessage.typService := LON_RESPONSE;
	typApplicationMessage.bSourceSubnetId := InDataTelegram_Module_1[1];
	typApplicationMessage.bSourceNodeId := InDataTelegram_Module_1[2];
	typApplicationMessage.bCorrelator := 0;
	typApplicationMessage.bCode :=  InDataTelegram_Module_1[3];
	typApplicationMessage.bDataLength := UINT_TO_BYTE(unLastLen_mbxModule_1 - 4);
	IF typApplicationMessage.bDataLength > 48 THEN typApplicationMessage.bDataLength := 48; END_IF;
	FuMemSet(ADR(typApplicationMessage.abData), 0, SIZEOF(typApplicationMessage.abData));
	IF typApplicationMessage.bDataLength > 0 THEN
		FuMemCopy(ADR(InDataTelegram_Module_1[4]), ADR(typApplicationMessage.abData), typApplicationMessage.bDataLength);
	END_IF
	typApplicationMessage.xRspRcvd := TRUE;
END_IF
END_ACTION
ACTION DomainDataRcvd:
IF (unLastLen_mbxModule_1 = 17) THEN
	iDomainTable := InDataTelegram_Module_1[1];
	IF (iDomainTable < 0) OR (iDomainTable > 1) THEN RETURN; END_IF
	FuMemCopy(ADR(InDataTelegram_Module_1[2]), ADR(atypDomainData[iDomainTable].abDomainId), 6);
	atypDomainData[iDomainTable].bSubnet := InDataTelegram_Module_1[8];
	atypDomainData[iDomainTable].xIsNonClone := InDataTelegram_Module_1[9].7;
	atypDomainData[iDomainTable].bNodeId := InDataTelegram_Module_1[9] AND 16#7F;
	atypDomainData[iDomainTable].xIsInvalid := InDataTelegram_Module_1[10].7;
	atypDomainData[iDomainTable].bDomainIdLength := InDataTelegram_Module_1[10] AND 16#7F;
	FuMemCopy(ADR(InDataTelegram_Module_1[11]), ADR(atypDomainData[iDomainTable].abAuthenticationKey), 6);
END_IF
END_ACTION
ACTION NeuronStateRcvd:
IF (unLastLen_mbxModule_1 = 16) THEN
	typNeuronState.wCrcError := InDataTelegram_Module_1[1] + InDataTelegram_Module_1[2] * 256;
	typNeuronState.wTransactionTimeouts := InDataTelegram_Module_1[3] + InDataTelegram_Module_1[4] * 256;
	typNeuronState.wReceiveTransactionBuffersFull := InDataTelegram_Module_1[5] + InDataTelegram_Module_1[6] * 256;
	typNeuronState.wLostMessages := InDataTelegram_Module_1[7] + InDataTelegram_Module_1[8] * 256;
	typNeuronState.wMissedMessages := InDataTelegram_Module_1[9] + InDataTelegram_Module_1[10] * 256;
	typNeuronState.bResetCause := InDataTelegram_Module_1[11];
	typNeuronState.bNodeState := InDataTelegram_Module_1[12];
	typNeuronState.bFirmwareVersion := InDataTelegram_Module_1[13];
	typNeuronState.bLastErrorLogged := InDataTelegram_Module_1[14];
	typNeuronState.bModelNumber := InDataTelegram_Module_1[15];
END_IF
END_ACTION
ACTION RequestNeuronState:
OutDataTelegram_Module_1[0] := C2M_MICRO_SERVER_STATUS_QRY;
OutDataTelegram_Module_1[1] := BOOL_TO_BYTE(trigReset.Q);

mbxModule_1.bTxPrio := 1;
mbxModule_1.bTxProtID := 0;
mbxModule_1.pbTxData := ADR(OutDataTelegram_Module_1);
mbxModule_1.unTxLen := 2;
mbxModule_1.MBX_SEND();

IF (mbxModule_1.nError <> MBX_OK) THEN
	RETURN;
END_IF
END_ACTION
ACTION ResetNviUpdate:
Module_1_PRG.SFPTnodeObject.ResetNviUpdate();
Module_1_PRG.Virtualfunctionalblock.ResetNviUpdate();
END_ACTION
ACTION SetParameter:
lonCom.pMbx 			:= ADR(mbxModule_1);
lonCom.pInData 			:= ADR(InDataTelegram_Module_1);
lonCom.pOutData 		:= ADR(OutDataTelegram_Module_1);
lonCom.pTimer			:= ADR(TimeoutTimer);

lonCom.pActualSignature	:= ADR(abSignature_Module_1);
lonCom.pConfigBlock := ADR(abInterface_Module_1);
lonCom.wConfigSize 		:= wConfigSize_Module_1;
END_ACTION

(* POU LON/Module_1/NV_Interface/Module_1_SFPTnodeObject, ST *)
FUNCTION_BLOCK Module_1_SFPTnodeObject
(******************************************)
(* Automatic generated code, do not edit! *)
(******************************************)
VAR_INPUT
	bObjectIndex : BYTE := 0;
	nvoStatus : typSnvtObjStatus;
	nvoFileStat : typSnvtFileStatus;

END_VAR
VAR_OUTPUT
	nviRequest : typSnvtObjRequest;
	nviFileReq : typSnvtFileReq;
	nviFilePos : typSnvtFilePos;

END_VAR
VAR
	xSetOnce : BOOL := TRUE;
	xDataInUpdated : BOOL := FALSE;
	nvoStatusLast: typSnvtObjStatus;
	nvoFileStatLast: typSnvtFileStatus;

	cmd : BYTE;
	z : INT;
	bNvRelativeIdx : BYTE;
	bNvAbsoluteIdx : BYTE;
	wCpRelativeIdx : WORD;
	wCpAbsoluteIdx : WORD;
END_VAR
VAR CONSTANT
	bNvStartIndex : BYTE := 0;
	wCpStartIndex : WORD := 65535;
	bLmoCount : BYTE := 1;
END_VAR
IF (xInitRunning_Module_1 = TRUE) AND (xSetOnce = TRUE) THEN
	xSetOnce := FALSE;
	CachePointers();
	SetUpdateFlags();
END_IF

CheckUpdateFlags();
IF (xInitRunning_Module_1 = FALSE) AND (xDataInUpdated = FALSE) THEN
	IF (mbxModule_1.bStatus.0) THEN
		SendValueRequest();
	END_IF
END_IF

IF (xInitRunning_Module_1 = FALSE) AND (mbxModule_1.bStatus.0) THEN
	xSetOnce := TRUE;
	xDataInUpdated := FALSE;
	IF ((NOT FuMemCompare(ADR(nvoStatusLast), ADR(nvoStatus), ADR(nvoStatus.bStatusInformation) - ADR(nvoStatus))) OR (nvoStatus.bStatusInformation.7 = TRUE) OR (nvoStatusLast.bInternalUseOnly.1 = TRUE)) THEN
		FuSnvtObjStatusToRaw(ADR(nvoStatus), ADR(OutDataTelegram_Module_1[2]));

		bNvAbsoluteIdx := bNvStartIndex + bObjectIndex + (1 * bLmoCount);

		IF (FuDoNvoUpdate_Module_1(ADR(nvoStatus), ADR(nvoStatusLast), ADR(nvoStatus.bInternalUseOnly), ADR(nvoStatusLast.bInternalUseOnly), ADR(nvoStatus.bStatusInformation), bNvAbsoluteIdx, 6, SIZEOF(nvoStatus)) = FALSE) THEN
			RETURN;
		END_IF
	END_IF
	IF ((NOT FuMemCompare(ADR(nvoFileStatLast), ADR(nvoFileStat), ADR(nvoFileStat.bStatusInformation) - ADR(nvoFileStat))) OR (nvoFileStat.bStatusInformation.7 = TRUE) OR (nvoFileStatLast.bInternalUseOnly.1 = TRUE)) THEN
		FuSnvtFileStatusToRaw(ADR(nvoFileStat), ADR(OutDataTelegram_Module_1[2]));

		bNvAbsoluteIdx := bNvStartIndex + bObjectIndex + (3 * bLmoCount);

		IF (FuDoNvoUpdate_Module_1(ADR(nvoFileStat), ADR(nvoFileStatLast), ADR(nvoFileStat.bInternalUseOnly), ADR(nvoFileStatLast.bInternalUseOnly), ADR(nvoFileStat.bStatusInformation), bNvAbsoluteIdx, 27, SIZEOF(nvoFileStat)) = FALSE) THEN
			RETURN;
		END_IF
	END_IF

END_IF
END_FUNCTION_BLOCK
ACTION CachePointers:
;
END_ACTION
ACTION CheckUpdateFlags:
xDataInUpdated := (NOT nviRequest.bInternalUseOnly.0) AND (NOT nviFileReq.bInternalUseOnly.0) AND (NOT nviFilePos.bInternalUseOnly.0) AND TRUE;
END_ACTION
ACTION DataReceived:
cmd := InDataTelegram_Module_1[0];
IF (cmd = M2C_NVI_UPDT_OCCD) OR (cmd = M2C_NV_VALUE_RSP) OR (cmd = M2C_NVI_UPDT_TOUT) THEN
	bNvRelativeIdx := (InDataTelegram_Module_1[1] - bNvStartIndex - bObjectIndex) / bLmoCount;
	CASE bNvRelativeIdx OF
	0:
		IF (cmd = M2C_NVI_UPDT_OCCD) OR (cmd = M2C_NV_VALUE_RSP) THEN
			IF (unLastLen_mbxModule_1 = (2 + 3)) THEN
				FuRawToSnvtObjRequest(ADR(InDataTelegram_Module_1[2]), ADR(nviRequest));
				nviRequest.bInternalUseOnly.0 := FALSE;
				nviRequest.bStatusInformation := FuInkrementNviStatus(nviRequest.bStatusInformation);
			ELSIF (unLastLen_mbxModule_1 = 2) THEN
				nviRequest.bStatusInformation := FuInkrementNviStatus(nviRequest.bStatusInformation);
			END_IF
		ELSIF (cmd = M2C_NVI_UPDT_TOUT) THEN
			IF (unLastLen_mbxModule_1 = 3) THEN
				nviRequest.bStatusInformation.4 := BYTE_TO_BOOL(InDataTelegram_Module_1[2]);
			END_IF
		END_IF
	2:
		IF (cmd = M2C_NVI_UPDT_OCCD) OR (cmd = M2C_NV_VALUE_RSP) THEN
			IF (unLastLen_mbxModule_1 = (2 + 12)) THEN
				FuRawToSnvtFileReq(ADR(InDataTelegram_Module_1[2]), ADR(nviFileReq));
				nviFileReq.bInternalUseOnly.0 := FALSE;
				nviFileReq.bStatusInformation := FuInkrementNviStatus(nviFileReq.bStatusInformation);
			ELSIF (unLastLen_mbxModule_1 = 2) THEN
				nviFileReq.bStatusInformation := FuInkrementNviStatus(nviFileReq.bStatusInformation);
			END_IF
		ELSIF (cmd = M2C_NVI_UPDT_TOUT) THEN
			IF (unLastLen_mbxModule_1 = 3) THEN
				nviFileReq.bStatusInformation.4 := BYTE_TO_BOOL(InDataTelegram_Module_1[2]);
			END_IF
		END_IF
	4:
		IF (cmd = M2C_NVI_UPDT_OCCD) OR (cmd = M2C_NV_VALUE_RSP) THEN
			IF (unLastLen_mbxModule_1 = (2 + 6)) THEN
				FuRawToSnvtFilePos(ADR(InDataTelegram_Module_1[2]), ADR(nviFilePos));
				nviFilePos.bInternalUseOnly.0 := FALSE;
				nviFilePos.bStatusInformation := FuInkrementNviStatus(nviFilePos.bStatusInformation);
			ELSIF (unLastLen_mbxModule_1 = 2) THEN
				nviFilePos.bStatusInformation := FuInkrementNviStatus(nviFilePos.bStatusInformation);
			END_IF
		ELSIF (cmd = M2C_NVI_UPDT_TOUT) THEN
			IF (unLastLen_mbxModule_1 = 3) THEN
				nviFilePos.bStatusInformation.4 := BYTE_TO_BOOL(InDataTelegram_Module_1[2]);
			END_IF
		END_IF

	END_CASE
ELSIF (cmd = M2C_CP_VALUE_RSP) THEN
	wCpRelativeIdx := ((InDataTelegram_Module_1[1] + InDataTelegram_Module_1[2] * 256) - wCpStartIndex - bObjectIndex) / bLmoCount;
	CASE wCpRelativeIdx OF

	END_CASE
END_IF
END_ACTION
ACTION ResetNviUpdate:
nviRequest.bStatusInformation := nviRequest.bStatusInformation AND 16#F8;
nviFileReq.bStatusInformation := nviFileReq.bStatusInformation AND 16#F8;
nviFilePos.bStatusInformation := nviFilePos.bStatusInformation AND 16#F8;
;
END_ACTION
ACTION SendValueRequest:
IF (FuSendNviValueReq_Module_1(ADR(nviRequest.bInternalUseOnly), bNvStartIndex + bObjectIndex + (0 * bLmoCount)) = FALSE) THEN
	RETURN;
END_IF

IF (FuSendNviValueReq_Module_1(ADR(nviFileReq.bInternalUseOnly), bNvStartIndex + bObjectIndex + (2 * bLmoCount)) = FALSE) THEN
	RETURN;
END_IF

IF (FuSendNviValueReq_Module_1(ADR(nviFilePos.bInternalUseOnly), bNvStartIndex + bObjectIndex + (4 * bLmoCount)) = FALSE) THEN
	RETURN;
END_IF

;
END_ACTION
ACTION SetUpdateFlags:
nviRequest.bInternaluseOnly.0 := TRUE;
nvoStatusLast.bInternaluseOnly.1 := TRUE;
nvoStatusLast.bInternaluseOnly.7 := FALSE;
nviFileReq.bInternaluseOnly.0 := TRUE;
nvoFileStatLast.bInternaluseOnly.1 := TRUE;
nvoFileStatLast.bInternaluseOnly.7 := FALSE;
nviFilePos.bInternaluseOnly.0 := TRUE;
;
END_ACTION

(* POU LON/Shared/Internal/FuSnvtObjStatusToRaw, ST *)
FUNCTION FuSnvtObjStatusToRaw : BOOL
(******************************************)
(* Automatic generated code, do not edit! *)
(******************************************)
VAR_INPUT
	NvDataIn :  POINTER TO typSnvtObjStatus;
	DataOut : POINTER TO ARRAY[0..5] OF BYTE;
END_VAR
VAR
END_VAR
DataOut^[0] := WORD_TO_BYTE(SHR(NvDataIn^.wObjectId, 8));
DataOut^[1] := WORD_TO_BYTE(NvDataIn^.wObjectId);

DataOut^[2] := NvDataIn^.bBitfieldByteOffset2;

DataOut^[3] := NvDataIn^.bBitfieldByteOffset3;

DataOut^[4] := NvDataIn^.bBitfieldByteOffset4;

DataOut^[5] := NvDataIn^.bBitfieldByteOffset5;

FuSnvtObjStatusToRaw := TRUE;
END_FUNCTION

(* POU LON/Module_1/Internal/FuDoNvoUpdate_Module_1, ST *)
FUNCTION FuDoNvoUpdate_Module_1 : BOOL
(******************************************)
(* Automatic generated code, do not edit! *)
(******************************************)
VAR_INPUT
	ptNvo : POINTER TO BYTE;
	ptNvoLast : POINTER TO BYTE;
	ptNvoInternalUse : POINTER TO BYTE;
	ptNvoLastInternalUse : POINTER TO BYTE;
	ptNvoStatusInformation : POINTER TO BYTE;
	bNvoIndex : BYTE;
	uiNvoLength : UINT;
	uiNvoVariableLength : UINT;
END_VAR
IF (ptNvoLastInternalUse^.1 = TRUE) AND (ptNvoStatusInformation^.7 = FALSE) THEN
	OutDataTelegram_Module_1[0] := C2M_NV_VALUE;
ELSE
	OutDataTelegram_Module_1[0] := C2M_NVO_PROPAGATE;
END_IF
OutDataTelegram_Module_1[1] := bNvoIndex;

mbxModule_1.bTxPrio := BOOL_TO_BYTE(ptNvoLastInternalUse^.7);
mbxModule_1.bTxProtID := 0;
mbxModule_1.pbTxData := ADR(OutDataTelegram_Module_1);
mbxModule_1.unTxLen := 2 + uiNvoLength;
mbxModule_1.MBX_SEND();

IF (mbxModule_1.nError <> MBX_OK) THEN
	FuDoNvoUpdate_Module_1 := FALSE;
	RETURN;
END_IF

ptNvoLastInternalUse^.1 := FALSE;
ptNvoInternalUse^ := ptNvoLastInternalUse^;
FuMemCopy(ptNvo, ptNvoLast, uiNvoVariableLength);

FuDoNvoUpdate_Module_1 := TRUE;
END_FUNCTION

(* POU LON/Shared/Internal/FuSnvtFileStatusToRaw, ST *)
FUNCTION FuSnvtFileStatusToRaw : BOOL
(******************************************)
(* Automatic generated code, do not edit! *)
(******************************************)
VAR_INPUT
	NvDataIn :  POINTER TO typSnvtFileStatus;
	DataOut : POINTER TO ARRAY[0..26] OF BYTE;
END_VAR
VAR
END_VAR
DataOut^[0] := NvDataIn^.bStatus;

DataOut^[1] := WORD_TO_BYTE(SHR(NvDataIn^.wNumberOfFiles, 8));
DataOut^[2] := WORD_TO_BYTE(NvDataIn^.wNumberOfFiles);

DataOut^[3] := WORD_TO_BYTE(SHR(NvDataIn^.wSelectedFile, 8));
DataOut^[4] := WORD_TO_BYTE(NvDataIn^.wSelectedFile);

DataOut^[5] := NvDataIn^.abAdr[0];
DataOut^[6] := NvDataIn^.abAdr[1];
DataOut^[7] := NvDataIn^.abAdr[2];
DataOut^[8] := NvDataIn^.abAdr[3];
DataOut^[9] := NvDataIn^.abAdr[4];
DataOut^[10] := NvDataIn^.abAdr[5];
DataOut^[11] := NvDataIn^.abAdr[6];
DataOut^[12] := NvDataIn^.abAdr[7];
DataOut^[13] := NvDataIn^.abAdr[8];
DataOut^[14] := NvDataIn^.abAdr[9];
DataOut^[15] := NvDataIn^.abAdr[10];
DataOut^[16] := NvDataIn^.abAdr[11];
DataOut^[17] := NvDataIn^.abAdr[12];
DataOut^[18] := NvDataIn^.abAdr[13];
DataOut^[19] := NvDataIn^.abAdr[14];
DataOut^[20] := NvDataIn^.abAdr[15];
DataOut^[21] := NvDataIn^.abAdr[16];
DataOut^[22] := NvDataIn^.abAdr[17];
DataOut^[23] := NvDataIn^.abAdr[18];
DataOut^[24] := NvDataIn^.abAdr[19];
DataOut^[25] := NvDataIn^.abAdr[20];
DataOut^[26] := NvDataIn^.abAdr[21];

FuSnvtFileStatusToRaw := TRUE;
END_FUNCTION

(* POU LON/Module_1/Internal/FuSendNviValueReq_Module_1, ST *)
FUNCTION FuSendNviValueReq_Module_1 : BOOL
(******************************************)
(* Automatic generated code, do not edit! *)
(******************************************)
VAR_INPUT
	ptInternalUseOnly : POINTER TO BYTE;
	bNvIndex : BYTE;
END_VAR
IF ptInternalUseOnly^.0 = TRUE THEN
	OutDataTelegram_Module_1[0] := C2M_NV_VALUE_QRY;
	OutDataTelegram_Module_1[1] := bNvIndex;

	mbxModule_1.bTxPrio := 1;
	mbxModule_1.bTxProtID := 0;
	mbxModule_1.pbTxData := ADR(OutDataTelegram_Module_1);
	mbxModule_1.unTxLen := 2;
	mbxModule_1.MBX_SEND();

	IF (mbxModule_1.nError <> MBX_OK) THEN
		FuSendNviValueReq_Module_1 := FALSE;
		RETURN;
	END_IF
	ptInternalUseOnly^.0 := FALSE;
END_IF

FuSendNviValueReq_Module_1 := TRUE;
END_FUNCTION

(* POU LON/Module_1/NV_Interface/Module_1_Virtualfunctionalblock, ST *)
FUNCTION_BLOCK Module_1_Virtualfunctionalblock
(******************************************)
(* Automatic generated code, do not edit! *)
(******************************************)
VAR_INPUT
	bObjectIndex : BYTE := 0;
	VT_Request : typSnvtObjRequest;
	VT_TimeSet : typSnvtTimeStamp;
	VT_AlarmSet : typSnvtAlarm;
	VT_HCC1_ModeSet : typSnvtHvacMode;
	VT_HCC1_TempSet : typSnvtTempP;
	VT_HCC1_SuppTemp : typSnvtTempP;
	VT_HCC2_ModeSet : typSnvtHvacMode;
	VT_HCC2_TempSet : typSnvtTempP;
	VT_HCC2_SuppTemp : typSnvtTempP;
	VT_HCC3_ModeSet : typSnvtHvacMode;
	VT_HCC3_TempSet : typSnvtTempP;
	VT_HCC3_SuppTemp : typSnvtTempP;
	VT_DHW_ModeSet : typSnvtHvacMode;
	VT_DHW_SetPoint : typSnvtTempP;
	VT_CFD_SetEnable : typSnvtSwitch;
	VT_CFD_SetMode : typSnvtHvacMode;
	VT_CFD_SetPoint : typSnvtTempP;

END_VAR
VAR_OUTPUT
	VT_Status : typSnvtObjStatus;
	VT_Alarm : typSnvtAlarm;
	VT_RlyState : typSnvtState;
	VT_HCC1_Mode : typSnvtHvacMode;
	VT_HCC1_Temp : typSnvtTempP;
	VT_HCC2_Mode : typSnvtHvacMode;
	VT_HCC2_Temp : typSnvtTempP;
	VT_HCC3_Mode : typSnvtHvacMode;
	VT_HCC3_Temp : typSnvtTempP;
	VT_DHW_ActTemp : typSnvtTempP;
	VT_DHW_TempSet : typSnvtTempP;
	VT_CFD_GetEnable : typSnvtSwitch;
	VT_CFD_Temp : typSnvtTempP;
	VT_CFD_SetTemp : typSnvtTempP;

END_VAR
VAR
	xSetOnce : BOOL := TRUE;
	xDataInUpdated : BOOL := FALSE;
	VT_RequestLast: typSnvtObjRequest;
	VT_TimeSetLast: typSnvtTimeStamp;
	VT_AlarmSetLast: typSnvtAlarm;
	VT_CFD_SetEnableLast: typSnvtSwitch;
	paNviSnvtHvacMode : ARRAY[0..2] OF POINTER TO typSnvtHvacMode;
	aNviSnvtHvacModeIndex : ARRAY[0..2] OF BYTE := 7,12,17;
	paNviSnvtTempP : ARRAY[0..6] OF POINTER TO typSnvtTempP;
	aNviSnvtTempPIndex : ARRAY[0..6] OF BYTE := 9,14,19,22,24,28,30;
	paNvoSnvtHvacMode : ARRAY[0..4] OF POINTER TO typSnvtHvacMode;
	aNvoSnvtHvacModeIndex : ARRAY[0..4] OF BYTE := 6,11,16,21,27;
	aNvoSnvtHvacModeLast : ARRAY[0..4] OF typSnvtHvacMode;
	aNvoSnvtHvacModePriority : ARRAY[0..0] OF BYTE := 16#00;
	paNvoSnvtTempP : ARRAY[0..7] OF POINTER TO typSnvtTempP;
	aNvoSnvtTempPIndex : ARRAY[0..7] OF BYTE := 8,10,13,15,18,20,23,29;
	aNvoSnvtTempPLast : ARRAY[0..7] OF typSnvtTempP;
	aNvoSnvtTempPPriority : ARRAY[0..0] OF BYTE := 16#00;

	cmd : BYTE;
	z : INT;
	bNvRelativeIdx : BYTE;
	bNvAbsoluteIdx : BYTE;
	wCpRelativeIdx : WORD;
	wCpAbsoluteIdx : WORD;
END_VAR
VAR CONSTANT
	bNvStartIndex : BYTE := 5;
	wCpStartIndex : WORD := 65535;
	bLmoCount : BYTE := 1;
END_VAR
IF (xInitRunning_Module_1 = TRUE) AND (xSetOnce = TRUE) THEN
	xSetOnce := FALSE;
	CachePointers();
	SetUpdateFlags();
END_IF

CheckUpdateFlags();
IF (xInitRunning_Module_1 = FALSE) AND (xDataInUpdated = FALSE) THEN
	IF (mbxModule_1.bStatus.0) THEN
		SendValueRequest();
	END_IF
END_IF

IF (xInitRunning_Module_1 = FALSE) AND (mbxModule_1.bStatus.0) THEN
	xSetOnce := TRUE;
	xDataInUpdated := FALSE;
	IF ((NOT FuMemCompare(ADR(VT_RequestLast), ADR(VT_Request), ADR(VT_Request.bStatusInformation) - ADR(VT_Request))) OR (VT_Request.bStatusInformation.7 = TRUE) OR (VT_RequestLast.bInternalUseOnly.1 = TRUE)) THEN
		FuSnvtObjRequestToRaw(ADR(VT_Request), ADR(OutDataTelegram_Module_1[2]));

		bNvAbsoluteIdx := bNvStartIndex + bObjectIndex + (0 * bLmoCount);

		IF (FuDoNvoUpdate_Module_1(ADR(VT_Request), ADR(VT_RequestLast), ADR(VT_Request.bInternalUseOnly), ADR(VT_RequestLast.bInternalUseOnly), ADR(VT_Request.bStatusInformation), bNvAbsoluteIdx, 3, SIZEOF(VT_Request)) = FALSE) THEN
			RETURN;
		END_IF
	END_IF
	IF ((NOT FuMemCompare(ADR(VT_TimeSetLast), ADR(VT_TimeSet), ADR(VT_TimeSet.bStatusInformation) - ADR(VT_TimeSet))) OR (VT_TimeSet.bStatusInformation.7 = TRUE) OR (VT_TimeSetLast.bInternalUseOnly.1 = TRUE)) THEN
		FuSnvtTimeStampToRaw(ADR(VT_TimeSet), ADR(OutDataTelegram_Module_1[2]));

		bNvAbsoluteIdx := bNvStartIndex + bObjectIndex + (2 * bLmoCount);

		IF (FuDoNvoUpdate_Module_1(ADR(VT_TimeSet), ADR(VT_TimeSetLast), ADR(VT_TimeSet.bInternalUseOnly), ADR(VT_TimeSetLast.bInternalUseOnly), ADR(VT_TimeSet.bStatusInformation), bNvAbsoluteIdx, 7, SIZEOF(VT_TimeSet)) = FALSE) THEN
			RETURN;
		END_IF
	END_IF
	IF ((NOT FuMemCompare(ADR(VT_AlarmSetLast), ADR(VT_AlarmSet), ADR(VT_AlarmSet.bStatusInformation) - ADR(VT_AlarmSet))) OR (VT_AlarmSet.bStatusInformation.7 = TRUE) OR (VT_AlarmSetLast.bInternalUseOnly.1 = TRUE)) THEN
		FuSnvtAlarmToRaw(ADR(VT_AlarmSet), ADR(OutDataTelegram_Module_1[2]));

		bNvAbsoluteIdx := bNvStartIndex + bObjectIndex + (4 * bLmoCount);

		IF (FuDoNvoUpdate_Module_1(ADR(VT_AlarmSet), ADR(VT_AlarmSetLast), ADR(VT_AlarmSet.bInternalUseOnly), ADR(VT_AlarmSetLast.bInternalUseOnly), ADR(VT_AlarmSet.bStatusInformation), bNvAbsoluteIdx, 29, SIZEOF(VT_AlarmSet)) = FALSE) THEN
			RETURN;
		END_IF
	END_IF
	IF ((NOT FuMemCompare(ADR(VT_CFD_SetEnableLast), ADR(VT_CFD_SetEnable), ADR(VT_CFD_SetEnable.bStatusInformation) - ADR(VT_CFD_SetEnable))) OR (VT_CFD_SetEnable.bStatusInformation.7 = TRUE) OR (VT_CFD_SetEnableLast.bInternalUseOnly.1 = TRUE)) THEN
		FuSnvtSwitchToRaw(ADR(VT_CFD_SetEnable), ADR(OutDataTelegram_Module_1[2]));

		bNvAbsoluteIdx := bNvStartIndex + bObjectIndex + (25 * bLmoCount);

		IF (FuDoNvoUpdate_Module_1(ADR(VT_CFD_SetEnable), ADR(VT_CFD_SetEnableLast), ADR(VT_CFD_SetEnable.bInternalUseOnly), ADR(VT_CFD_SetEnableLast.bInternalUseOnly), ADR(VT_CFD_SetEnable.bStatusInformation), bNvAbsoluteIdx, 2, SIZEOF(VT_CFD_SetEnable)) = FALSE) THEN
			RETURN;
		END_IF
	END_IF
	FOR z := 0 TO 4 DO
		IF ((NOT FuMemCompare(ADR(aNvoSnvtHvacModeLast[z]), paNvoSnvtHvacMode[z], ADR(paNvoSnvtHvacMode[z]^.bStatusInformation) - paNvoSnvtHvacMode[z])) OR (paNvoSnvtHvacMode[z]^.bStatusInformation.7 = TRUE) OR (aNvoSnvtHvacModeLast[z].bInternalUseOnly.1 = TRUE)) THEN
			FuSnvtHvacModeToRaw(paNvoSnvtHvacMode[z], ADR(OutDataTelegram_Module_1[2]));

			bNvAbsoluteIdx := bNvStartIndex + bObjectIndex + (aNvoSnvtHvacModeIndex[z] * bLmoCount);

			IF (FuDoNvoUpdate_Module_1(paNvoSnvtHvacMode[z], ADR(aNvoSnvtHvacModeLast[z]), ADR(paNvoSnvtHvacMode[z]^.bInternalUseOnly), ADR(aNvoSnvtHvacModeLast[z].bInternalUseOnly), ADR(paNvoSnvtHvacMode[z]^.bStatusInformation), bNvAbsoluteIdx, 1, SIZEOF(aNvoSnvtHvacModeLast[z])) = FALSE) THEN
				RETURN;
			END_IF
		END_IF
	END_FOR
	FOR z := 0 TO 7 DO
		IF ((NOT FuMemCompare(ADR(aNvoSnvtTempPLast[z]), paNvoSnvtTempP[z], ADR(paNvoSnvtTempP[z]^.bStatusInformation) - paNvoSnvtTempP[z])) OR (paNvoSnvtTempP[z]^.bStatusInformation.7 = TRUE) OR (aNvoSnvtTempPLast[z].bInternalUseOnly.1 = TRUE)) THEN
			FuSnvtTempPToRaw(paNvoSnvtTempP[z], ADR(OutDataTelegram_Module_1[2]));

			bNvAbsoluteIdx := bNvStartIndex + bObjectIndex + (aNvoSnvtTempPIndex[z] * bLmoCount);

			IF (FuDoNvoUpdate_Module_1(paNvoSnvtTempP[z], ADR(aNvoSnvtTempPLast[z]), ADR(paNvoSnvtTempP[z]^.bInternalUseOnly), ADR(aNvoSnvtTempPLast[z].bInternalUseOnly), ADR(paNvoSnvtTempP[z]^.bStatusInformation), bNvAbsoluteIdx, 2, SIZEOF(aNvoSnvtTempPLast[z])) = FALSE) THEN
				RETURN;
			END_IF
		END_IF
	END_FOR

END_IF
END_FUNCTION_BLOCK
ACTION CachePointers:
paNviSnvtHvacMode[0] := ADR(VT_HCC1_Mode);
paNviSnvtHvacMode[1] := ADR(VT_HCC2_Mode);
paNviSnvtHvacMode[2] := ADR(VT_HCC3_Mode);
paNviSnvtTempP[0] := ADR(VT_HCC1_Temp);
paNviSnvtTempP[1] := ADR(VT_HCC2_Temp);
paNviSnvtTempP[2] := ADR(VT_HCC3_Temp);
paNviSnvtTempP[3] := ADR(VT_DHW_ActTemp);
paNviSnvtTempP[4] := ADR(VT_DHW_TempSet);
paNviSnvtTempP[5] := ADR(VT_CFD_Temp);
paNviSnvtTempP[6] := ADR(VT_CFD_SetTemp);
paNvoSnvtHvacMode[0] := ADR(VT_HCC1_ModeSet);
paNvoSnvtHvacMode[1] := ADR(VT_HCC2_ModeSet);
paNvoSnvtHvacMode[2] := ADR(VT_HCC3_ModeSet);
paNvoSnvtHvacMode[3] := ADR(VT_DHW_ModeSet);
paNvoSnvtHvacMode[4] := ADR(VT_CFD_SetMode);
paNvoSnvtTempP[0] := ADR(VT_HCC1_TempSet);
paNvoSnvtTempP[1] := ADR(VT_HCC1_SuppTemp);
paNvoSnvtTempP[2] := ADR(VT_HCC2_TempSet);
paNvoSnvtTempP[3] := ADR(VT_HCC2_SuppTemp);
paNvoSnvtTempP[4] := ADR(VT_HCC3_TempSet);
paNvoSnvtTempP[5] := ADR(VT_HCC3_SuppTemp);
paNvoSnvtTempP[6] := ADR(VT_DHW_SetPoint);
paNvoSnvtTempP[7] := ADR(VT_CFD_SetPoint);
;
END_ACTION
ACTION CheckUpdateFlags:
xDataInUpdated := (NOT VT_Status.bInternalUseOnly.0) AND (NOT VT_Alarm.bInternalUseOnly.0) AND (NOT VT_RlyState.bInternalUseOnly.0) AND (NOT VT_CFD_GetEnable.bInternalUseOnly.0) AND TRUE;
FOR z := 0 TO 2 DO
	xDataInUpdated := xDataInUpdated AND (NOT paNviSnvtHvacMode[z]^.bInternalUseOnly.0);
END_FOR
FOR z := 0 TO 6 DO
	xDataInUpdated := xDataInUpdated AND (NOT paNviSnvtTempP[z]^.bInternalUseOnly.0);
END_FOR
END_ACTION
ACTION DataReceived:
cmd := InDataTelegram_Module_1[0];
IF (cmd = M2C_NVI_UPDT_OCCD) OR (cmd = M2C_NV_VALUE_RSP) OR (cmd = M2C_NVI_UPDT_TOUT) THEN
	bNvRelativeIdx := (InDataTelegram_Module_1[1] - bNvStartIndex - bObjectIndex) / bLmoCount;
	CASE bNvRelativeIdx OF
	1:
		IF (cmd = M2C_NVI_UPDT_OCCD) OR (cmd = M2C_NV_VALUE_RSP) THEN
			IF (unLastLen_mbxModule_1 = (2 + 6)) THEN
				FuRawToSnvtObjStatus(ADR(InDataTelegram_Module_1[2]), ADR(VT_Status));
				VT_Status.bInternalUseOnly.0 := FALSE;
				VT_Status.bStatusInformation := FuInkrementNviStatus(VT_Status.bStatusInformation);
			ELSIF (unLastLen_mbxModule_1 = 2) THEN
				VT_Status.bStatusInformation := FuInkrementNviStatus(VT_Status.bStatusInformation);
			END_IF
		ELSIF (cmd = M2C_NVI_UPDT_TOUT) THEN
			IF (unLastLen_mbxModule_1 = 3) THEN
				VT_Status.bStatusInformation.4 := BYTE_TO_BOOL(InDataTelegram_Module_1[2]);
			END_IF
		END_IF
	3:
		IF (cmd = M2C_NVI_UPDT_OCCD) OR (cmd = M2C_NV_VALUE_RSP) THEN
			IF (unLastLen_mbxModule_1 = (2 + 29)) THEN
				FuRawToSnvtAlarm(ADR(InDataTelegram_Module_1[2]), ADR(VT_Alarm));
				VT_Alarm.bInternalUseOnly.0 := FALSE;
				VT_Alarm.bStatusInformation := FuInkrementNviStatus(VT_Alarm.bStatusInformation);
			ELSIF (unLastLen_mbxModule_1 = 2) THEN
				VT_Alarm.bStatusInformation := FuInkrementNviStatus(VT_Alarm.bStatusInformation);
			END_IF
		ELSIF (cmd = M2C_NVI_UPDT_TOUT) THEN
			IF (unLastLen_mbxModule_1 = 3) THEN
				VT_Alarm.bStatusInformation.4 := BYTE_TO_BOOL(InDataTelegram_Module_1[2]);
			END_IF
		END_IF
	5:
		IF (cmd = M2C_NVI_UPDT_OCCD) OR (cmd = M2C_NV_VALUE_RSP) THEN
			IF (unLastLen_mbxModule_1 = (2 + 2)) THEN
				FuRawToSnvtState(ADR(InDataTelegram_Module_1[2]), ADR(VT_RlyState));
				VT_RlyState.bInternalUseOnly.0 := FALSE;
				VT_RlyState.bStatusInformation := FuInkrementNviStatus(VT_RlyState.bStatusInformation);
			ELSIF (unLastLen_mbxModule_1 = 2) THEN
				VT_RlyState.bStatusInformation := FuInkrementNviStatus(VT_RlyState.bStatusInformation);
			END_IF
		ELSIF (cmd = M2C_NVI_UPDT_TOUT) THEN
			IF (unLastLen_mbxModule_1 = 3) THEN
				VT_RlyState.bStatusInformation.4 := BYTE_TO_BOOL(InDataTelegram_Module_1[2]);
			END_IF
		END_IF
	26:
		IF (cmd = M2C_NVI_UPDT_OCCD) OR (cmd = M2C_NV_VALUE_RSP) THEN
			IF (unLastLen_mbxModule_1 = (2 + 2)) THEN
				FuRawToSnvtSwitch(ADR(InDataTelegram_Module_1[2]), ADR(VT_CFD_GetEnable));
				VT_CFD_GetEnable.bInternalUseOnly.0 := FALSE;
				VT_CFD_GetEnable.bStatusInformation := FuInkrementNviStatus(VT_CFD_GetEnable.bStatusInformation);
			ELSIF (unLastLen_mbxModule_1 = 2) THEN
				VT_CFD_GetEnable.bStatusInformation := FuInkrementNviStatus(VT_CFD_GetEnable.bStatusInformation);
			END_IF
		ELSIF (cmd = M2C_NVI_UPDT_TOUT) THEN
			IF (unLastLen_mbxModule_1 = 3) THEN
				VT_CFD_GetEnable.bStatusInformation.4 := BYTE_TO_BOOL(InDataTelegram_Module_1[2]);
			END_IF
		END_IF
	7, 12, 17:
		IF (cmd = M2C_NVI_UPDT_OCCD) OR (cmd = M2C_NV_VALUE_RSP) THEN
			IF (unLastLen_mbxModule_1 = (2 + 1)) THEN
				FOR z := 0 TO 2 DO
					IF aNviSnvtHvacModeIndex[z] = bNvRelativeIdx THEN
						FuRawToSnvtHvacMode(ADR(InDataTelegram_Module_1[2]), paNviSnvtHvacMode[z]);
						paNviSnvtHvacMode[z]^.bInternalUseOnly.0 := FALSE;
						paNviSnvtHvacMode[z]^.bStatusInformation := FuInkrementNviStatus(paNviSnvtHvacMode[z]^.bStatusInformation);
						EXIT;
					END_IF
				END_FOR
			ELSIF (unLastLen_mbxModule_1 = 2) THEN
				FOR z := 0 TO 2 DO
					IF aNviSnvtHvacModeIndex[z] = bNvRelativeIdx THEN
						paNviSnvtHvacMode[z]^.bStatusInformation := FuInkrementNviStatus(paNviSnvtHvacMode[z]^.bStatusInformation);
						EXIT;
					END_IF
				END_FOR
			END_IF
		ELSIF (cmd = M2C_NVI_UPDT_TOUT) THEN
			IF (unLastLen_mbxModule_1 = 3) THEN
				FOR z := 0 TO 2 DO
					IF aNviSnvtHvacModeIndex[z] = bNvRelativeIdx THEN
						paNviSnvtHvacMode[z]^.bStatusInformation.4 := BYTE_TO_BOOL(InDataTelegram_Module_1[2]);
						EXIT;
					END_IF
				END_FOR
			END_IF
		END_IF
	9, 14, 19, 22, 24, 28, 30:
		IF (cmd = M2C_NVI_UPDT_OCCD) OR (cmd = M2C_NV_VALUE_RSP) THEN
			IF (unLastLen_mbxModule_1 = (2 + 2)) THEN
				FOR z := 0 TO 6 DO
					IF aNviSnvtTempPIndex[z] = bNvRelativeIdx THEN
						FuRawToSnvtTempP(ADR(InDataTelegram_Module_1[2]), paNviSnvtTempP[z]);
						paNviSnvtTempP[z]^.bInternalUseOnly.0 := FALSE;
						paNviSnvtTempP[z]^.bStatusInformation := FuInkrementNviStatus(paNviSnvtTempP[z]^.bStatusInformation);
						EXIT;
					END_IF
				END_FOR
			ELSIF (unLastLen_mbxModule_1 = 2) THEN
				FOR z := 0 TO 6 DO
					IF aNviSnvtTempPIndex[z] = bNvRelativeIdx THEN
						paNviSnvtTempP[z]^.bStatusInformation := FuInkrementNviStatus(paNviSnvtTempP[z]^.bStatusInformation);
						EXIT;
					END_IF
				END_FOR
			END_IF
		ELSIF (cmd = M2C_NVI_UPDT_TOUT) THEN
			IF (unLastLen_mbxModule_1 = 3) THEN
				FOR z := 0 TO 6 DO
					IF aNviSnvtTempPIndex[z] = bNvRelativeIdx THEN
						paNviSnvtTempP[z]^.bStatusInformation.4 := BYTE_TO_BOOL(InDataTelegram_Module_1[2]);
						EXIT;
					END_IF
				END_FOR
			END_IF
		END_IF

	END_CASE
ELSIF (cmd = M2C_CP_VALUE_RSP) THEN
	wCpRelativeIdx := ((InDataTelegram_Module_1[1] + InDataTelegram_Module_1[2] * 256) - wCpStartIndex - bObjectIndex) / bLmoCount;
	CASE wCpRelativeIdx OF

	END_CASE
END_IF
END_ACTION
ACTION ResetNviUpdate:
VT_Status.bStatusInformation := VT_Status.bStatusInformation AND 16#F8;
VT_Alarm.bStatusInformation := VT_Alarm.bStatusInformation AND 16#F8;
VT_RlyState.bStatusInformation := VT_RlyState.bStatusInformation AND 16#F8;
VT_CFD_GetEnable.bStatusInformation := VT_CFD_GetEnable.bStatusInformation AND 16#F8;
FOR z := 0 TO 2 DO
	paNviSnvtHvacMode[z]^.bStatusInformation := paNviSnvtHvacMode[z]^.bStatusInformation AND 16#F8;
END_FOR
FOR z := 0 TO 6 DO
	paNviSnvtTempP[z]^.bStatusInformation := paNviSnvtTempP[z]^.bStatusInformation AND 16#F8;
END_FOR
;
END_ACTION
ACTION SendValueRequest:
IF (FuSendNviValueReq_Module_1(ADR(VT_Status.bInternalUseOnly), bNvStartIndex + bObjectIndex + (1 * bLmoCount)) = FALSE) THEN
	RETURN;
END_IF

IF (FuSendNviValueReq_Module_1(ADR(VT_Alarm.bInternalUseOnly), bNvStartIndex + bObjectIndex + (3 * bLmoCount)) = FALSE) THEN
	RETURN;
END_IF

IF (FuSendNviValueReq_Module_1(ADR(VT_RlyState.bInternalUseOnly), bNvStartIndex + bObjectIndex + (5 * bLmoCount)) = FALSE) THEN
	RETURN;
END_IF

IF (FuSendNviValueReq_Module_1(ADR(VT_CFD_GetEnable.bInternalUseOnly), bNvStartIndex + bObjectIndex + (26 * bLmoCount)) = FALSE) THEN
	RETURN;
END_IF

FOR z := 0 TO 2 DO
	IF (FuSendNviValueReq_Module_1(ADR(paNviSnvtHvacMode[z]^.bInternalUseOnly), bNvStartIndex + bObjectIndex + (aNviSnvtHvacModeIndex[z] * bLmoCount)) = FALSE) THEN
		RETURN;
	END_IF;
END_FOR;
FOR z := 0 TO 6 DO
	IF (FuSendNviValueReq_Module_1(ADR(paNviSnvtTempP[z]^.bInternalUseOnly), bNvStartIndex + bObjectIndex + (aNviSnvtTempPIndex[z] * bLmoCount)) = FALSE) THEN
		RETURN;
	END_IF;
END_FOR;
;
END_ACTION
ACTION SetUpdateFlags:
VT_RequestLast.bInternaluseOnly.1 := TRUE;
VT_RequestLast.bInternaluseOnly.7 := FALSE;
VT_Status.bInternaluseOnly.0 := TRUE;
VT_TimeSetLast.bInternaluseOnly.1 := TRUE;
VT_TimeSetLast.bInternaluseOnly.7 := FALSE;
VT_Alarm.bInternaluseOnly.0 := TRUE;
VT_AlarmSetLast.bInternaluseOnly.1 := TRUE;
VT_AlarmSetLast.bInternaluseOnly.7 := FALSE;
VT_RlyState.bInternaluseOnly.0 := TRUE;
VT_CFD_SetEnableLast.bInternaluseOnly.1 := TRUE;
VT_CFD_SetEnableLast.bInternaluseOnly.7 := FALSE;
VT_CFD_GetEnable.bInternaluseOnly.0 := TRUE;
FOR z := 0 TO 2 DO
	paNviSnvtHvacMode[z]^.bInternaluseOnly.0 := TRUE;
END_FOR;
FOR z := 0 TO 6 DO
	paNviSnvtTempP[z]^.bInternaluseOnly.0 := TRUE;
END_FOR;
FOR z := 0 TO 4 DO
	aNvoSnvtHvacModeLast[z].bInternaluseOnly.1 := TRUE;
	aNvoSnvtHvacModeLast[z].bInternaluseOnly.7 := (SHR(aNvoSnvtHvacModePriority[z / 8], z MOD 8) AND 1) <> 0;
END_FOR;
FOR z := 0 TO 7 DO
	aNvoSnvtTempPLast[z].bInternaluseOnly.1 := TRUE;
	aNvoSnvtTempPLast[z].bInternaluseOnly.7 := (SHR(aNvoSnvtTempPPriority[z / 8], z MOD 8) AND 1) <> 0;
END_FOR;
;
END_ACTION

(* POU LON/Shared/Internal/FuSnvtObjRequestToRaw, ST *)
FUNCTION FuSnvtObjRequestToRaw : BOOL
(******************************************)
(* Automatic generated code, do not edit! *)
(******************************************)
VAR_INPUT
	NvDataIn :  POINTER TO typSnvtObjRequest;
	DataOut : POINTER TO ARRAY[0..2] OF BYTE;
END_VAR
VAR
END_VAR
DataOut^[0] := WORD_TO_BYTE(SHR(NvDataIn^.wObjectId, 8));
DataOut^[1] := WORD_TO_BYTE(NvDataIn^.wObjectId);

DataOut^[2] := NvDataIn^.bObjectRequest;

FuSnvtObjRequestToRaw := TRUE;
END_FUNCTION

(* POU LON/Shared/Internal/FuSnvtTimeStampToRaw, ST *)
FUNCTION FuSnvtTimeStampToRaw : BOOL
(******************************************)
(* Automatic generated code, do not edit! *)
(******************************************)
VAR_INPUT
	NvDataIn :  POINTER TO typSnvtTimeStamp;
	DataOut : POINTER TO ARRAY[0..6] OF BYTE;
END_VAR
VAR
END_VAR
DataOut^[0] := INT_TO_BYTE(SHR(NvDataIn^.iYear, 8));
DataOut^[1] := INT_TO_BYTE(NvDataIn^.iYear);

DataOut^[2] := NvDataIn^.bMonth;

DataOut^[3] := NvDataIn^.bDay;

DataOut^[4] := NvDataIn^.bHour;

DataOut^[5] := NvDataIn^.bMinute;

DataOut^[6] := NvDataIn^.bSecond;

FuSnvtTimeStampToRaw := TRUE;
END_FUNCTION

(* POU LON/Shared/Internal/FuSnvtAlarmToRaw, ST *)
FUNCTION FuSnvtAlarmToRaw : BOOL
(******************************************)
(* Automatic generated code, do not edit! *)
(******************************************)
VAR_INPUT
	NvDataIn :  POINTER TO typSnvtAlarm;
	DataOut : POINTER TO ARRAY[0..28] OF BYTE;
END_VAR
VAR
END_VAR
DataOut^[0] := NvDataIn^.abLocation[0];
DataOut^[1] := NvDataIn^.abLocation[1];
DataOut^[2] := NvDataIn^.abLocation[2];
DataOut^[3] := NvDataIn^.abLocation[3];
DataOut^[4] := NvDataIn^.abLocation[4];
DataOut^[5] := NvDataIn^.abLocation[5];

DataOut^[6] := WORD_TO_BYTE(SHR(NvDataIn^.wObjectId, 8));
DataOut^[7] := WORD_TO_BYTE(NvDataIn^.wObjectId);

DataOut^[8] := NvDataIn^.bAlarmType;

DataOut^[9] := NvDataIn^.bPriorityLevel;

DataOut^[10] := WORD_TO_BYTE(SHR(NvDataIn^.wIndexToSnvt, 8));
DataOut^[11] := WORD_TO_BYTE(NvDataIn^.wIndexToSnvt);

DataOut^[12] := NvDataIn^.abValue[0];
DataOut^[13] := NvDataIn^.abValue[1];
DataOut^[14] := NvDataIn^.abValue[2];
DataOut^[15] := NvDataIn^.abValue[3];

DataOut^[16] := WORD_TO_BYTE(SHR(NvDataIn^.wYear, 8));
DataOut^[17] := WORD_TO_BYTE(NvDataIn^.wYear);

DataOut^[18] := NvDataIn^.bMonth;

DataOut^[19] := NvDataIn^.bDay;

DataOut^[20] := NvDataIn^.bHour;

DataOut^[21] := NvDataIn^.bMinute;

DataOut^[22] := NvDataIn^.bSecond;

DataOut^[23] := WORD_TO_BYTE(SHR(NvDataIn^.wMillisecond, 8));
DataOut^[24] := WORD_TO_BYTE(NvDataIn^.wMillisecond);

DataOut^[25] := NvDataIn^.abAlarmLimit[0];
DataOut^[26] := NvDataIn^.abAlarmLimit[1];
DataOut^[27] := NvDataIn^.abAlarmLimit[2];
DataOut^[28] := NvDataIn^.abAlarmLimit[3];

FuSnvtAlarmToRaw := TRUE;
END_FUNCTION

(* POU LON/Shared/Internal/FuSnvtSwitchToRaw, ST *)
FUNCTION FuSnvtSwitchToRaw : BOOL
(******************************************)
(* Automatic generated code, do not edit! *)
(******************************************)
VAR_INPUT
	NvDataIn :  POINTER TO typSnvtSwitch;
	DataOut : POINTER TO ARRAY[0..1] OF BYTE;
END_VAR
VAR
END_VAR
DataOut^[0] := NvDataIn^.bValue;

DataOut^[1] := NvDataIn^.siState;

FuSnvtSwitchToRaw := TRUE;
END_FUNCTION

(* POU LON/Shared/Internal/FuSnvtHvacModeToRaw, ST *)
FUNCTION FuSnvtHvacModeToRaw : BOOL
(******************************************)
(* Automatic generated code, do not edit! *)
(******************************************)
VAR_INPUT
	NvDataIn :  POINTER TO typSnvtHvacMode;
	DataOut : POINTER TO ARRAY[0..0] OF BYTE;
END_VAR
VAR
END_VAR
DataOut^[0] := NvDataIn^.bSnvtHvacMode;

FuSnvtHvacModeToRaw := TRUE;
END_FUNCTION

(* POU LON/Shared/Internal/FuSnvtTempPToRaw, ST *)
FUNCTION FuSnvtTempPToRaw : BOOL
(******************************************)
(* Automatic generated code, do not edit! *)
(******************************************)
VAR_INPUT
	NvDataIn :  POINTER TO typSnvtTempP;
	DataOut : POINTER TO ARRAY[0..1] OF BYTE;
END_VAR
VAR
END_VAR
DataOut^[0] := INT_TO_BYTE(SHR(NvDataIn^.iSnvtTempP, 8));
DataOut^[1] := INT_TO_BYTE(NvDataIn^.iSnvtTempP);

FuSnvtTempPToRaw := TRUE;
END_FUNCTION

(* POU TCP_Logger/Logger_Proc, ST *)
PROGRAM Logger_Proc
VAR
	c1:         	TCPCLIENT;

	Open:	    	BOOL;
	IpAddr:			DWORD;
	InetAddr:		DWORD;
	Connected:  	BOOL;
	Error:      	DINT;
	TxTrig:     	BOOL;
	RxData:			ARRAY [0..MAX_RECEIVE_TCP_CLIENT] OF BYTE;
	RxLen:			DINT;

	Retry:			BYTE;	(* Counter for connection retries *)
	Recovered:		BYTE;	(* Counter for recovered unsent messages *)

	i:				DINT;
	pos:			DWORD;
	hFile:			DWORD;

END_VAR
(*=== State machine ===*)
CASE Logger.Status OF

	S_Logger_UNKNOWN:
		(* Startup *)
		Logger.SendReq:=FALSE;
		Open:=FALSE;
		Logger.Status:=S_Logger_IDLE;

	S_Logger_IDLE:
		(* Wait request *)
		IF Logger.SendReq THEN
			(* Resolve server name or use static IP *)
			IF LEN(Logger_SERVER)=0 THEN
				InetAddr:=SysSockInetAddr(Logger_IP);
			ELSE
				IpAddr:=SysSockGetHostByName(ADR(Logger_SERVER));
				DWORDSWAP(pIn:=ADR(IpAddr), pOut:=ADR(InetAddr));
			END_IF
			TxTrig:=FALSE;
			RxLen:=0;
			(* Open connection *)
			Open:=TRUE;
			Logger.Status:=S_Logger_WAITCONN;
		END_IF

	S_Logger_WAITCONN:
		(* Wait connection *)
		IF Connected THEN
			(* Send data *)
			TxTrig:=TRUE;
			Logger.Status:=S_Logger_WAITTX;
		END_IF
		IF Error>0 THEN
			Open:=FALSE;
			Logger.Status:=S_Logger_ERROR;
		END_IF

	S_Logger_WAITTX:
		(* Wait transmission *)
		IF NOT TxTrig THEN
			Logger.Status:=S_Logger_WAITRESP;
		END_IF
		IF Error>0 THEN
			Open:=FALSE;
			Logger.Status:=S_Logger_ERROR;
		END_IF

	S_Logger_WAITRESP:
		(* Wait response *)
		IF Connected=FALSE (* OR TIMEOUT!! *) THEN
			Open:=FALSE;
			(* Check response *)
			IF RxLen>=4 AND CHKSTRING(pString:=ADR(RxData), pPattern:=ADR(Logger_CHECK)) THEN
				Logger.SendReq:=FALSE;
				Retry:=0;
				(* Check unsent messages to flush *)
				IF Recovered<Logger_RecoverMsgs THEN
					MsgChk();
					IF Logger.SendReq=TRUE THEN
						Recovered:=Recovered+1;
					ELSE
						Recovered:=0;
					END_IF
				ELSE
					Recovered:=0;
				END_IF
				Logger.Status:=S_Logger_IDLE;
			ELSE
				Logger.Status:=S_Logger_ERROR;
			END_IF
		END_IF

